LIN {X 0,Y 468.2,Z 260.249,A -85,B 0,C 180,E1 -7618.306,E2 -7618.306} C_VEL
LIN {X 0,Y 467.957,Z 265.306,A -85,B 0,C 180,E1 -7620.584,E2 -7620.584} C_VEL
LIN {X 0,Y 467.636,Z 273.513,A -85,B 0,C 180,E1 -7624.161,E2 -7624.161} C_VEL
LIN {X 0,Y 467.386,Z 281.282,A -85,B 0,C 180,E1 -7627.453,E2 -7627.453} C_VEL
LIN {X 0,Y 467.175,Z 287.892,A -85,B 0,C 180,E1 -7630.215,E2 -7630.215} C_VEL
LIN {X 0,Y 467.029,Z 295.543,A -85,B 0,C 180,E1 -7633.386,E2 -7633.386} C_VEL
LIN {X 0,Y 466.937,Z 298.461,A -85,B 0,C 180,E1 -7634.594,E2 -7634.594} C_VEL
LIN {X 0,Y 469.237,Z 312.548,A -85,B 0,C 180,E1 -7635.056,E2 -7635.056} C_VEL
LIN {X 0,Y 469.965,Z 320.318,A -85,B 0,C 180,E1 -7635.383,E2 -7635.383} C_VEL
LIN {X 0,Y 469.517,Z 331.349,A -85,B 0,C 180,E1 -7635.922,E2 -7635.922} C_VEL
LIN {X 0,Y 469.015,Z 343.205,A -85,B 0,C 180,E1 -7636.68,E2 -7636.68} C_VEL
LIN {X 0,Y 468.525,Z 353.704,A -85,B 0,C 180,E1 -7637.535,E2 -7637.535} C_VEL
LIN {X 0,Y 468.12,Z 363.549,A -85,B 0,C 180,E1 -7638.526,E2 -7638.526} C_VEL
LIN {X 0,Y 467.618,Z 372.397,A -85,B 0,C 180,E1 -7639.61,E2 -7639.61} C_VEL
LIN {X 0,Y 467.263,Z 381.03,A -85,B 0,C 180,E1 -7640.913,E2 -7640.913} C_VEL
LIN {X 0,Y 466.991,Z 387.93,A -85,B 0,C 180,E1 -7642.215,E2 -7642.215} C_VEL
LIN {X 0,Y 466.816,Z 393.538,A -85,B 0,C 180,E1 -7643.537,E2 -7643.537} C_VEL
LIN {X 0,Y 466.737,Z 397.799,A -85,B 0,C 180,E1 -7644.816,E2 -7644.816} C_VEL
LIN {X 0,Y 466.647,Z 400.094,A -85,B 0,C 180,E1 -7645.681,E2 -7645.681} C_VEL
LIN {X 0,Y 466.689,Z 401.958,A -85,B 0,C 180,E1 -7646.546,E2 -7646.546} C_VEL
LIN {X 0,Y 466.662,Z 403.353,A -85,B 0,C 180,E1 -7647.41,E2 -7647.41} C_VEL
LIN {X 0,Y 466.618,Z 404.957,A -85,B 0,C 180,E1 -7649.137,E2 -7649.137} C_VEL
LIN {X 0,Y 466.598,Z 405.173,A -85,B 0,C 180,E1 -7650,E2 -7650} C_VEL
LIN {X 0,Y 466.618,Z 404.957,A -85,B 0,C 180,E1 -7650.863,E2 -7650.863} C_VEL
LIN {X 0,Y 466.662,Z 403.356,A -85,B 0,C 180,E1 -7652.589,E2 -7652.589} C_VEL
LIN {X 0,Y 466.689,Z 401.961,A -85,B 0,C 180,E1 -7653.453,E2 -7653.453} C_VEL
LIN {X 0,Y 466.689,Z 399.024,A -85,B 0,C 180,E1 -7654.751,E2 -7654.751} C_VEL
LIN {X 0,Y 466.755,Z 395.05,A -85,B 0,C 180,E1 -7656.05,E2 -7656.05} C_VEL
LIN {X 0,Y 466.971,Z 388.941,A -85,B 0,C 180,E1 -7657.567,E2 -7657.567} C_VEL
LIN {X 0,Y 467.227,Z 382.264,A -85,B 0,C 180,E1 -7658.869,E2 -7658.869} C_VEL
LIN {X 0,Y 467.565,Z 373.98,A -85,B 0,C 180,E1 -7660.173,E2 -7660.173} C_VEL
LIN {X 0,Y 468.023,Z 365.492,A -85,B 0,C 180,E1 -7661.257,E2 -7661.257} C_VEL
LIN {X 0,Y 468.46,Z 355.447,A -85,B 0,C 180,E1 -7662.303,E2 -7662.303} C_VEL
LIN {X 0,Y 468.941,Z 344.625,A -85,B 0,C 180,E1 -7663.212,E2 -7663.212} C_VEL
LIN {X 0,Y 469.441,Z 333.25,A -85,B 0,C 180,E1 -7663.97,E2 -7663.97} C_VEL
LIN {X 0,Y 469.914,Z 321.583,A -85,B 0,C 180,E1 -7664.563,E2 -7664.563} C_VEL
LIN {X 0,Y 469.724,Z 316.487,A -85,B 0,C 180,E1 -7664.783,E2 -7664.783} C_VEL
LIN {X 0,Y 467.709,Z 303.026,A -85,B 0,C 180,E1 -7665.271,E2 -7665.271} C_VEL
LIN {X 0,Y 466.937,Z 298.457,A -85,B 0,C 180,E1 -7665.406,E2 -7665.406} C_VEL
LIN {X 0,Y 467.114,Z 290.788,A -85,B 0,C 180,E1 -7668.581,E2 -7668.581} C_VEL
LIN {X 0,Y 467.347,Z 283.49,A -85,B 0,C 180,E1 -7671.619,E2 -7671.619} C_VEL
LIN {X 0,Y 467.56,Z 275.713,A -85,B 0,C 180,E1 -7674.89,E2 -7674.89} C_VEL
LIN {X 0,Y 467.794,Z 267.942,A -85,B 0,C 180,E1 -7678.245,E2 -7678.245} C_VEL
LIN {X 0,Y 468.087,Z 262.432,A -85,B 0,C 180,E1 -7680.696,E2 -7680.696} C_VEL
LIN {X 0,Y 468.438,Z 255.839,A -85,B 0,C 180,E1 -7683.719,E2 -7683.719} C_VEL
LIN {X 0,Y 468.486,Z 251.281,A -85,B 0,C 180,E1 -7685.896,E2 -7685.896} C_VEL
LIN {X 0,Y 467.682,Z 245.54,A -85,B 0,C 180,E1 -7688.834,E2 -7688.834} C_VEL
LIN {X 0,Y 467.621,Z 245.24,A -85,B 0,C 180,E1 -7689.141,E2 -7689.141} C_VEL
LIN {X 0,Y 467.588,Z 245.241,A -85,B 0,C 180,E1 -7692.567,E2 -7692.567} C_VEL
LIN {X 0,Y 467.567,Z 245.245,A -85,B 0,C 180,E1 -7695.052,E2 -7695.052} C_VEL
LIN {X 0,Y 467.566,Z 245.246,A -85,B 0,C 180,E1 -7698.725,E2 -7698.725} C_VEL
LIN {X 0,Y 467.562,Z 245.242,A -85,B 0,C 180,E1 -7701.955,E2 -7701.955} C_VEL
LIN {X 0,Y 467.564,Z 245.243,A -85,B 0,C 180,E1 -7705.167,E2 -7705.167} C_VEL
LIN {X 0,Y 467.585,Z 245.241,A -85,B 0,C 180,E1 -7708.26,E2 -7708.26} C_VEL
LIN {X 0,Y 467.555,Z 245.244,A -85,B 0,C 180,E1 -7711.249,E2 -7711.249} C_VEL
LIN {X 0,Y 467.568,Z 245.246,A -85,B 0,C 180,E1 -7714.157,E2 -7714.157} C_VEL
LIN {X 0,Y 467.577,Z 245.239,A -85,B 0,C 180,E1 -7716.996,E2 -7716.996} C_VEL
LIN {X 0,Y 467.625,Z 245.238,A -85,B 0,C 180,E1 -7719.777,E2 -7719.777} C_VEL
LIN {X 0,Y 467.609,Z 245.239,A -85,B 0,C 180,E1 -7722.507,E2 -7722.507} C_VEL
LIN {X 0,Y 467.605,Z 245.238,A -85,B 0,C 180,E1 -7725.196,E2 -7725.196} C_VEL
LIN {X 0,Y 467.657,Z 245.235,A -85,B 0,C 180,E1 -7727.855,E2 -7727.855} C_VEL
LIN {X 0,Y 467.668,Z 245.232,A -85,B 0,C 180,E1 -7731.357,E2 -7731.357} C_VEL
LIN {X 0,Y 467.736,Z 245.221,A -85,B 0,C 180,E1 -7733.963,E2 -7733.963} C_VEL
LIN {X 0,Y 467.861,Z 245.206,A -85,B 0,C 180,E1 -7737.417,E2 -7737.417} C_VEL
LIN {X 0,Y 467.882,Z 245.204,A -85,B 0,C 180,E1 -7740,E2 -7740} C_VEL
LIN {X 0,Y 467.822,Z 245.21,A -85,B 0,C 180,E1 -7742.583,E2 -7742.583} C_VEL
LIN {X 0,Y 467.725,Z 245.22,A -85,B 0,C 180,E1 -7746.038,E2 -7746.038} C_VEL
LIN {X 0,Y 467.673,Z 245.232,A -85,B 0,C 180,E1 -7748.643,E2 -7748.643} C_VEL
LIN {X 0,Y 467.658,Z 245.232,A -85,B 0,C 180,E1 -7752.145,E2 -7752.145} C_VEL
LIN {X 0,Y 467.64,Z 245.233,A -85,B 0,C 180,E1 -7755.695,E2 -7755.695} C_VEL
LIN {X 0,Y 467.623,Z 245.234,A -85,B 0,C 180,E1 -7759.308,E2 -7759.308} C_VEL
LIN {X 0,Y 467.537,Z 245.247,A -85,B 0,C 180,E1 -7762.074,E2 -7762.074} C_VEL
LIN {X 0,Y 467.588,Z 245.24,A -85,B 0,C 180,E1 -7764.888,E2 -7764.888} C_VEL
LIN {X 0,Y 467.621,Z 245.238,A -85,B 0,C 180,E1 -7767.769,E2 -7767.769} C_VEL
LIN {X 0,Y 467.568,Z 245.242,A -85,B 0,C 180,E1 -7771.045,E2 -7771.045} C_VEL
LIN {X 0,Y 467.578,Z 245.244,A -85,B 0,C 180,E1 -7774.24,E2 -7774.24} C_VEL
LIN {X 0,Y 467.545,Z 245.244,A -85,B 0,C 180,E1 -7777.186,E2 -7777.186} C_VEL
LIN {X 0,Y 467.574,Z 245.242,A -85,B 0,C 180,E1 -7780.265,E2 -7780.265} C_VEL
LIN {X 0,Y 467.549,Z 245.245,A -85,B 0,C 180,E1 -7783.745,E2 -7783.745} C_VEL
LIN {X 0,Y 467.533,Z 245.248,A -85,B 0,C 180,E1 -7786.253,E2 -7786.253} C_VEL
LIN {X 0,Y 467.559,Z 245.246,A -85,B 0,C 180,E1 -7789.733,E2 -7789.733} C_VEL
LIN {X 0,Y 467.54,Z 245.248,A -85,B 0,C 180,E1 -7792.815,E2 -7792.815} C_VEL
LIN {X 0,Y 467.465,Z 245.257,A -85,B 0,C 180,E1 -7794.278,E2 -7794.278} C_VEL
LIN {X 0,Y 467.468,Z 246.827,A -85,B 0,C 180,E1 -7795.78,E2 -7795.78} C_VEL
LIN {X 0,Y 467.357,Z 251.614,A -85,B 0,C 180,E1 -7799.251,E2 -7799.251} C_VEL
LIN {X 0,Y 467.182,Z 255.798,A -85,B 0,C 180,E1 -7802.203,E2 -7802.203} C_VEL
LIN {X 0,Y 467.117,Z 259.954,A -85,B 0,C 180,E1 -7805.085,E2 -7805.085} C_VEL
LIN {X 0,Y 466.987,Z 264.104,A -85,B 0,C 180,E1 -7807.899,E2 -7807.899} C_VEL
LIN {X 0,Y 466.904,Z 269.34,A -85,B 0,C 180,E1 -7811.322,E2 -7811.322} C_VEL
LIN {X 0,Y 466.827,Z 273.108,A -85,B 0,C 180,E1 -7813.712,E2 -7813.712} C_VEL
LIN {X 0,Y 466.726,Z 274.503,A -85,B 0,C 180,E1 -7814.089,E2 -7814.089} C_VEL
LIN {X 0,Y 466.338,Z 277.681,A -85,B 0,C 180,E1 -7814.465,E2 -7814.465} C_VEL
LIN {X 0,Y 465.543,Z 283.2,A -85,B 0,C 180,E1 -7814.816,E2 -7814.816} C_VEL
LIN {X 0,Y 463.983,Z 293.781,A -85,B 0,C 180,E1 -7815.189,E2 -7815.189} C_VEL
LIN {X 0,Y 463.138,Z 301.031,A -85,B 0,C 180,E1 -7815.502,E2 -7815.502} C_VEL
LIN {X 0,Y 462.696,Z 312.356,A -85,B 0,C 180,E1 -7816.159,E2 -7816.159} C_VEL
LIN {X 0,Y 462.211,Z 324.024,A -85,B 0,C 180,E1 -7817.04,E2 -7817.04} C_VEL
LIN {X 0,Y 461.626,Z 334.493,A -85,B 0,C 180,E1 -7818.028,E2 -7818.028} C_VEL
LIN {X 0,Y 461.182,Z 343.044,A -85,B 0,C 180,E1 -7819.019,E2 -7819.019} C_VEL
LIN {X 0,Y 460.763,Z 350.92,A -85,B 0,C 180,E1 -7820.119,E2 -7820.119} C_VEL
LIN {X 0,Y 460.321,Z 358.62,A -85,B 0,C 180,E1 -7821.439,E2 -7821.439} C_VEL
LIN {X 0,Y 460.003,Z 365.682,A -85,B 0,C 180,E1 -7822.98,E2 -7822.98} C_VEL
LIN {X 0,Y 459.88,Z 370.386,A -85,B 0,C 180,E1 -7824.299,E2 -7824.299} C_VEL
LIN {X 0,Y 459.679,Z 373.991,A -85,B 0,C 180,E1 -7825.616,E2 -7825.616} C_VEL
LIN {X 0,Y 459.689,Z 375.851,A -85,B 0,C 180,E1 -7826.494,E2 -7826.494} C_VEL
LIN {X 0,Y 459.607,Z 377.256,A -85,B 0,C 180,E1 -7827.371,E2 -7827.371} C_VEL
LIN {X 0,Y 459.523,Z 378.87,A -85,B 0,C 180,E1 -7829.124,E2 -7829.124} C_VEL
LIN {X 0,Y 459.531,Z 379.105,A -85,B 0,C 180,E1 -7830,E2 -7830} C_VEL
LIN {X 0,Y 459.523,Z 378.919,A -85,B 0,C 180,E1 -7830.876,E2 -7830.876} C_VEL
LIN {X 0,Y 459.607,Z 377.369,A -85,B 0,C 180,E1 -7832.629,E2 -7832.629} C_VEL
LIN {X 0,Y 459.688,Z 376.013,A -85,B 0,C 180,E1 -7833.506,E2 -7833.506} C_VEL
LIN {X 0,Y 459.67,Z 373.152,A -85,B 0,C 180,E1 -7834.824,E2 -7834.824} C_VEL
LIN {X 0,Y 459.941,Z 369.265,A -85,B 0,C 180,E1 -7836.14,E2 -7836.14} C_VEL
LIN {X 0,Y 460.051,Z 364.257,A -85,B 0,C 180,E1 -7837.461,E2 -7837.461} C_VEL
LIN {X 0,Y 460.361,Z 357.95,A -85,B 0,C 180,E1 -7838.781,E2 -7838.781} C_VEL
LIN {X 0,Y 460.782,Z 350.052,A -85,B 0,C 180,E1 -7840.102,E2 -7840.102} C_VEL
LIN {X 0,Y 461.299,Z 340.226,A -85,B 0,C 180,E1 -7841.424,E2 -7841.424} C_VEL
LIN {X 0,Y 461.897,Z 329.928,A -85,B 0,C 180,E1 -7842.521,E2 -7842.521} C_VEL
LIN {X 0,Y 462.402,Z 318.607,A -85,B 0,C 180,E1 -7843.489,E2 -7843.489} C_VEL
LIN {X 0,Y 462.943,Z 306.706,A -85,B 0,C 180,E1 -7844.282,E2 -7844.282} C_VEL
LIN {X 0,Y 463.324,Z 294.664,A -85,B 0,C 180,E1 -7844.887,E2 -7844.887} C_VEL
LIN {X 0,Y 462.666,Z 288.508,A -85,B 0,C 180,E1 -7845.158,E2 -7845.158} C_VEL
LIN {X 0,Y 459.907,Z 275.491,A -85,B 0,C 180,E1 -7845.643,E2 -7845.643} C_VEL
LIN {X 0,Y 459.836,Z 274.771,A -85,B 0,C 180,E1 -7845.704,E2 -7845.704} C_VEL
LIN {X 0,Y 459.843,Z 270.048,A -85,B 0,C 180,E1 -7848.721,E2 -7848.721} C_VEL
LIN {X 0,Y 459.908,Z 265.809,A -85,B 0,C 180,E1 -7851.516,E2 -7851.516} C_VEL
LIN {X 0,Y 460.008,Z 261.63,A -85,B 0,C 180,E1 -7854.363,E2 -7854.363} C_VEL
LIN {X 0,Y 460.133,Z 256.956,A -85,B 0,C 180,E1 -7857.639,E2 -7857.639} C_VEL
LIN {X 0,Y 460.231,Z 253.27,A -85,B 0,C 180,E1 -7860.261,E2 -7860.261} C_VEL
LIN {X 0,Y 460.349,Z 249.051,A -85,B 0,C 180,E1 -7863.34,E2 -7863.34} C_VEL
LIN {X 0,Y 460.367,Z 246.221,A -85,B 0,C 180,E1 -7865.459,E2 -7865.459} C_VEL
LIN {X 0,Y 460.499,Z 246.122,A -85,B 0,C 180,E1 -7867.624,E2 -7867.624} C_VEL
LIN {X 0,Y 460.518,Z 246.12,A -85,B 0,C 180,E1 -7871.013,E2 -7871.013} C_VEL
LIN {X 0,Y 460.512,Z 246.122,A -85,B 0,C 180,E1 -7874.59,E2 -7874.59} C_VEL
LIN {X 0,Y 460.506,Z 246.123,A -85,B 0,C 180,E1 -7877.816,E2 -7877.816} C_VEL
LIN {X 0,Y 460.536,Z 246.117,A -85,B 0,C 180,E1 -7881.104,E2 -7881.104} C_VEL
LIN {X 0,Y 460.511,Z 246.12,A -85,B 0,C 180,E1 -7884.554,E2 -7884.554} C_VEL
LIN {X 0,Y 460.532,Z 246.122,A -85,B 0,C 180,E1 -7887.715,E2 -7887.715} C_VEL
LIN {X 0,Y 460.54,Z 246.118,A -85,B 0,C 180,E1 -7890.769,E2 -7890.769} C_VEL
LIN {X 0,Y 460.559,Z 246.116,A -85,B 0,C 180,E1 -7893.734,E2 -7893.734} C_VEL
LIN {X 0,Y 460.548,Z 246.116,A -85,B 0,C 180,E1 -7896.624,E2 -7896.624} C_VEL
LIN {X 0,Y 460.554,Z 246.119,A -85,B 0,C 180,E1 -7899.453,E2 -7899.453} C_VEL
LIN {X 0,Y 460.543,Z 246.117,A -85,B 0,C 180,E1 -7902.229,E2 -7902.229} C_VEL
LIN {X 0,Y 460.565,Z 246.118,A -85,B 0,C 180,E1 -7904.965,E2 -7904.965} C_VEL
LIN {X 0,Y 460.615,Z 246.11,A -85,B 0,C 180,E1 -7908.559,E2 -7908.559} C_VEL
LIN {X 0,Y 460.624,Z 246.11,A -85,B 0,C 180,E1 -7911.224,E2 -7911.224} C_VEL
LIN {X 0,Y 460.693,Z 246.096,A -85,B 0,C 180,E1 -7913.87,E2 -7913.87} C_VEL
LIN {X 0,Y 460.767,Z 246.089,A -85,B 0,C 180,E1 -7917.377,E2 -7917.377} C_VEL
LIN {X 0,Y 460.825,Z 246.083,A -85,B 0,C 180,E1 -7920,E2 -7920} C_VEL
LIN {X 0,Y 460.803,Z 246.086,A -85,B 0,C 180,E1 -7922.622,E2 -7922.622} C_VEL
LIN {X 0,Y 460.703,Z 246.097,A -85,B 0,C 180,E1 -7926.13,E2 -7926.13} C_VEL
LIN {X 0,Y 460.61,Z 246.11,A -85,B 0,C 180,E1 -7928.776,E2 -7928.776} C_VEL
LIN {X 0,Y 460.599,Z 246.112,A -85,B 0,C 180,E1 -7932.435,E2 -7932.435} C_VEL
LIN {X 0,Y 460.604,Z 246.112,A -85,B 0,C 180,E1 -7935.997,E2 -7935.997} C_VEL
LIN {X 0,Y 460.574,Z 246.114,A -85,B 0,C 180,E1 -7938.902,E2 -7938.902} C_VEL
LIN {X 0,Y 460.519,Z 246.12,A -85,B 0,C 180,E1 -7941.486,E2 -7941.486} C_VEL
LIN {X 0,Y 460.52,Z 246.12,A -85,B 0,C 180,E1 -7944.334,E2 -7944.334} C_VEL
LIN {X 0,Y 460.531,Z 246.119,A -85,B 0,C 180,E1 -7947.247,E2 -7947.247} C_VEL
LIN {X 0,Y 460.509,Z 246.123,A -85,B 0,C 180,E1 -7950.24,E2 -7950.24} C_VEL
LIN {X 0,Y 460.532,Z 246.12,A -85,B 0,C 180,E1 -7953.325,E2 -7953.325} C_VEL
LIN {X 0,Y 460.475,Z 246.125,A -85,B 0,C 180,E1 -7956.53,E2 -7956.53} C_VEL
LIN {X 0,Y 460.515,Z 246.12,A -85,B 0,C 180,E1 -7959.864,E2 -7959.864} C_VEL
LIN {X 0,Y 460.482,Z 246.127,A -85,B 0,C 180,E1 -7962.896,E2 -7962.896} C_VEL
LIN {X 0,Y 460.511,Z 246.123,A -85,B 0,C 180,E1 -7965.831,E2 -7965.831} C_VEL
LIN {X 0,Y 460.533,Z 246.121,A -85,B 0,C 180,E1 -7968.989,E2 -7968.989} C_VEL
LIN {X 0,Y 460.605,Z 246.235,A -85,B 0,C 180,E1 -7970.847,E2 -7970.847} C_VEL
LIN {X 0,Y 461.46,Z 251.948,A -85,B 0,C 180,E1 -7973.822,E2 -7973.822} C_VEL
LIN {X 0,Y 461.425,Z 256.864,A -85,B 0,C 180,E1 -7976.225,E2 -7976.225} C_VEL
LIN {X 0,Y 461.058,Z 264.541,A -85,B 0,C 180,E1 -7979.799,E2 -7979.799} C_VEL
LIN {X 0,Y 460.648,Z 272.27,A -85,B 0,C 180,E1 -7983.251,E2 -7983.251} C_VEL
LIN {X 0,Y 460.39,Z 279.379,A -85,B 0,C 180,E1 -7986.337,E2 -7986.337} C_VEL
LIN {X 0,Y 460.204,Z 286.63,A -85,B 0,C 180,E1 -7989.436,E2 -7989.436} C_VEL
LIN {X 0,Y 459.965,Z 294.285,A -85,B 0,C 180,E1 -7992.665,E2 -7992.665} C_VEL
LIN {X 0,Y 459.85,Z 298.232,A -85,B 0,C 180,E1 -7994.333,E2 -7994.333} C_VEL
LIN {X 0,Y 462.417,Z 313.883,A -85,B 0,C 180,E1 -7994.887,E2 -7994.887} C_VEL
LIN {X 0,Y 463.043,Z 321.426,A -85,B 0,C 180,E1 -7995.216,E2 -7995.216} C_VEL
LIN {X 0,Y 462.528,Z 333.073,A -85,B 0,C 180,E1 -7995.817,E2 -7995.817} C_VEL
LIN {X 0,Y 462.02,Z 344.438,A -85,B 0,C 180,E1 -7996.587,E2 -7996.587} C_VEL
LIN {X 0,Y 461.506,Z 355.549,A -85,B 0,C 180,E1 -7997.536,E2 -7997.536} C_VEL
LIN {X 0,Y 461.061,Z 365.301,A -85,B 0,C 180,E1 -7998.57,E2 -7998.57} C_VEL
LIN {X 0,Y 460.522,Z 373.785,A -85,B 0,C 180,E1 -7999.67,E2 -7999.67} C_VEL
LIN {X 0,Y 460.159,Z 382.067,A -85,B 0,C 180,E1 -8000.993,E2 -8000.993} C_VEL
LIN {X 0,Y 459.888,Z 388.743,A -85,B 0,C 180,E1 -8002.315,E2 -8002.315} C_VEL
LIN {X 0,Y 459.671,Z 394.853,A -85,B 0,C 180,E1 -8003.856,E2 -8003.856} C_VEL
LIN {X 0,Y 459.617,Z 398.825,A -85,B 0,C 180,E1 -8005.176,E2 -8005.176} C_VEL
LIN {X 0,Y 459.584,Z 401.758,A -85,B 0,C 180,E1 -8006.493,E2 -8006.493} C_VEL
LIN {X 0,Y 459.584,Z 403.154,A -85,B 0,C 180,E1 -8007.37,E2 -8007.37} C_VEL
LIN {X 0,Y 459.521,Z 404.757,A -85,B 0,C 180,E1 -8009.124,E2 -8009.124} C_VEL
LIN {X 0,Y 459.53,Z 404.974,A -85,B 0,C 180,E1 -8010,E2 -8010} C_VEL
LIN {X 0,Y 459.521,Z 404.757,A -85,B 0,C 180,E1 -8010.876,E2 -8010.876} C_VEL
LIN {X 0,Y 459.584,Z 403.156,A -85,B 0,C 180,E1 -8012.629,E2 -8012.629} C_VEL
LIN {X 0,Y 459.584,Z 401.76,A -85,B 0,C 180,E1 -8013.507,E2 -8013.507} C_VEL
LIN {X 0,Y 459.617,Z 398.824,A -85,B 0,C 180,E1 -8014.824,E2 -8014.824} C_VEL
LIN {X 0,Y 459.714,Z 393.819,A -85,B 0,C 180,E1 -8016.431,E2 -8016.431} C_VEL
LIN {X 0,Y 459.932,Z 387.726,A -85,B 0,C 180,E1 -8017.905,E2 -8017.905} C_VEL
LIN {X 0,Y 460.23,Z 380.824,A -85,B 0,C 180,E1 -8019.227,E2 -8019.227} C_VEL
LIN {X 0,Y 460.602,Z 372.189,A -85,B 0,C 180,E1 -8020.55,E2 -8020.55} C_VEL
LIN {X 0,Y 461.141,Z 363.339,A -85,B 0,C 180,E1 -8021.65,E2 -8021.65} C_VEL
LIN {X 0,Y 461.644,Z 352.452,A -85,B 0,C 180,E1 -8022.752,E2 -8022.752} C_VEL
LIN {X 0,Y 462.148,Z 341.45,A -85,B 0,C 180,E1 -8023.634,E2 -8023.634} C_VEL
LIN {X 0,Y 462.717,Z 329.129,A -85,B 0,C 180,E1 -8024.401,E2 -8024.401} C_VEL
LIN {X 0,Y 462.995,Z 318.768,A -85,B 0,C 180,E1 -8024.898,E2 -8024.898} C_VEL
LIN {X 0,Y 461.197,Z 306.142,A -85,B 0,C 180,E1 -8025.406,E2 -8025.406} C_VEL
LIN {X 0,Y 459.85,Z 298.222,A -85,B 0,C 180,E1 -8025.667,E2 -8025.667} C_VEL
LIN {X 0,Y 460.053,Z 291.009,A -85,B 0,C 180,E1 -8028.712,E2 -8028.712} C_VEL
LIN {X 0,Y 460.299,Z 283.333,A -85,B 0,C 180,E1 -8031.967,E2 -8031.967} C_VEL
LIN {X 0,Y 460.535,Z 275.574,A -85,B 0,C 180,E1 -8035.296,E2 -8035.296} C_VEL
LIN {X 0,Y 460.864,Z 267.822,A -85,B 0,C 180,E1 -8038.709,E2 -8038.709} C_VEL
LIN {X 0,Y 461.147,Z 261.894,A -85,B 0,C 180,E1 -8041.41,E2 -8041.41} C_VEL
LIN {X 0,Y 461.511,Z 254.948,A -85,B 0,C 180,E1 -8044.682,E2 -8044.682} C_VEL
LIN {X 0,Y 461.228,Z 250.3,A -85,B 0,C 180,E1 -8047.005,E2 -8047.005} C_VEL
LIN {X 0,Y 460.572,Z 246.118,A -85,B 0,C 180,E1 -8049.219,E2 -8049.219} C_VEL
LIN {X 0,Y 460.524,Z 246.126,A -85,B 0,C 180,E1 -8052.181,E2 -8052.181} C_VEL
LIN {X 0,Y 460.513,Z 246.125,A -85,B 0,C 180,E1 -8055.411,E2 -8055.411} C_VEL
LIN {X 0,Y 460.519,Z 246.122,A -85,B 0,C 180,E1 -8058.987,E2 -8058.987} C_VEL
LIN {X 0,Y 460.499,Z 246.127,A -85,B 0,C 180,E1 -8062.377,E2 -8062.377} C_VEL
LIN {X 0,Y 460.547,Z 246.117,A -85,B 0,C 180,E1 -8065.624,E2 -8065.624} C_VEL
LIN {X 0,Y 460.539,Z 246.121,A -85,B 0,C 180,E1 -8068.745,E2 -8068.745} C_VEL
LIN {X 0,Y 460.551,Z 246.119,A -85,B 0,C 180,E1 -8072.261,E2 -8072.261} C_VEL
LIN {X 0,Y 460.523,Z 246.119,A -85,B 0,C 180,E1 -8074.703,E2 -8074.703} C_VEL
LIN {X 0,Y 460.512,Z 246.122,A -85,B 0,C 180,E1 -8077.571,E2 -8077.571} C_VEL
LIN {X 0,Y 460.571,Z 246.114,A -85,B 0,C 180,E1 -8080.385,E2 -8080.385} C_VEL
LIN {X 0,Y 460.566,Z 246.116,A -85,B 0,C 180,E1 -8083.146,E2 -8083.146} C_VEL
LIN {X 0,Y 460.553,Z 246.118,A -85,B 0,C 180,E1 -8085.868,E2 -8085.868} C_VEL
LIN {X 0,Y 460.608,Z 246.108,A -85,B 0,C 180,E1 -8088.559,E2 -8088.559} C_VEL
LIN {X 0,Y 460.618,Z 246.109,A -85,B 0,C 180,E1 -8091.224,E2 -8091.224} C_VEL
LIN {X 0,Y 460.701,Z 246.097,A -85,B 0,C 180,E1 -8093.87,E2 -8093.87} C_VEL
LIN {X 0,Y 460.802,Z 246.086,A -85,B 0,C 180,E1 -8097.378,E2 -8097.378} C_VEL
LIN {X 0,Y 460.851,Z 246.079,A -85,B 0,C 180,E1 -8100,E2 -8100} C_VEL
LIN {X 0,Y 460.766,Z 246.089,A -85,B 0,C 180,E1 -8102.623,E2 -8102.623} C_VEL
LIN {X 0,Y 460.692,Z 246.096,A -85,B 0,C 180,E1 -8106.13,E2 -8106.13} C_VEL
LIN {X 0,Y 460.623,Z 246.111,A -85,B 0,C 180,E1 -8108.776,E2 -8108.776} C_VEL
LIN {X 0,Y 460.616,Z 246.111,A -85,B 0,C 180,E1 -8112.445,E2 -8112.445} C_VEL
LIN {X 0,Y 460.602,Z 246.111,A -85,B 0,C 180,E1 -8115.998,E2 -8115.998} C_VEL
LIN {X 0,Y 460.569,Z 246.112,A -85,B 0,C 180,E1 -8119.616,E2 -8119.616} C_VEL
LIN {X 0,Y 460.513,Z 246.124,A -85,B 0,C 180,E1 -8122.429,E2 -8122.429} C_VEL
LIN {X 0,Y 460.555,Z 246.117,A -85,B 0,C 180,E1 -8125.798,E2 -8125.798} C_VEL
LIN {X 0,Y 460.553,Z 246.117,A -85,B 0,C 180,E1 -8128.233,E2 -8128.233} C_VEL
LIN {X 0,Y 460.521,Z 246.12,A -85,B 0,C 180,E1 -8131.283,E2 -8131.283} C_VEL
LIN {X 0,Y 460.523,Z 246.12,A -85,B 0,C 180,E1 -8134.504,E2 -8134.504} C_VEL
LIN {X 0,Y 460.5,Z 246.124,A -85,B 0,C 180,E1 -8137.623,E2 -8137.623} C_VEL
LIN {X 0,Y 460.538,Z 246.118,A -85,B 0,C 180,E1 -8140.269,E2 -8140.269} C_VEL
LIN {X 0,Y 460.51,Z 246.123,A -85,B 0,C 180,E1 -8143.375,E2 -8143.375} C_VEL
LIN {X 0,Y 460.489,Z 246.124,A -85,B 0,C 180,E1 -8146.623,E2 -8146.623} C_VEL
LIN {X 0,Y 460.525,Z 246.122,A -85,B 0,C 180,E1 -8149.733,E2 -8149.733} C_VEL
LIN {X 0,Y 460.496,Z 246.123,A -85,B 0,C 180,E1 -8152.525,E2 -8152.525} C_VEL
LIN {X 0,Y 460.377,Z 246.142,A -85,B 0,C 180,E1 -8154.542,E2 -8154.542} C_VEL
LIN {X 0,Y 460.358,Z 249.508,A -85,B 0,C 180,E1 -8157.104,E2 -8157.104} C_VEL
LIN {X 0,Y 460.259,Z 253.124,A -85,B 0,C 180,E1 -8159.742,E2 -8159.742} C_VEL
LIN {X 0,Y 460.122,Z 257.314,A -85,B 0,C 180,E1 -8162.727,E2 -8162.727} C_VEL
LIN {X 0,Y 460.024,Z 261.487,A -85,B 0,C 180,E1 -8165.639,E2 -8165.639} C_VEL
LIN {X 0,Y 459.912,Z 266.098,A -85,B 0,C 180,E1 -8168.774,E2 -8168.774} C_VEL
LIN {X 0,Y 459.789,Z 271.312,A -85,B 0,C 180,E1 -8172.199,E2 -8172.199} C_VEL
LIN {X 0,Y 459.831,Z 274.824,A -85,B 0,C 180,E1 -8174.421,E2 -8174.421} C_VEL
LIN {X 0,Y 462.871,Z 289.702,A -85,B 0,C 180,E1 -8174.985,E2 -8174.985} C_VEL
LIN {X 0,Y 463.385,Z 293.828,A -85,B 0,C 180,E1 -8175.171,E2 -8175.171} C_VEL
LIN {X 0,Y 463.138,Z 301.031,A -85,B 0,C 180,E1 -8175.502,E2 -8175.502} C_VEL
LIN {X 0,Y 462.242,Z 306.474,A -85,B 0,C 180,E1 -8175.769,E2 -8175.769} C_VEL
LIN {X 0,Y 459.129,Z 315.145,A -85,B 0,C 180,E1 -8176.228,E2 -8176.228} C_VEL
LIN {X 0,Y 455.996,Z 323.415,A -85,B 0,C 180,E1 -8176.783,E2 -8176.783} C_VEL
LIN {X 0,Y 455.073,Z 328.224,A -85,B 0,C 180,E1 -8177.196,E2 -8177.196} C_VEL
LIN {X 0,Y 454.542,Z 337.717,A -85,B 0,C 180,E1 -8178.178,E2 -8178.178} C_VEL
LIN {X 0,Y 454.063,Z 346.563,A -85,B 0,C 180,E1 -8179.296,E2 -8179.296} C_VEL
LIN {X 0,Y 453.545,Z 355.194,A -85,B 0,C 180,E1 -8180.636,E2 -8180.636} C_VEL
LIN {X 0,Y 453.116,Z 362.075,A -85,B 0,C 180,E1 -8181.976,E2 -8181.976} C_VEL
LIN {X 0,Y 452.881,Z 367.544,A -85,B 0,C 180,E1 -8183.306,E2 -8183.306} C_VEL
LIN {X 0,Y 452.699,Z 371.904,A -85,B 0,C 180,E1 -8184.655,E2 -8184.655} C_VEL
LIN {X 0,Y 452.588,Z 374.192,A -85,B 0,C 180,E1 -8185.547,E2 -8185.547} C_VEL
LIN {X 0,Y 452.607,Z 376.052,A -85,B 0,C 180,E1 -8186.439,E2 -8186.439} C_VEL
LIN {X 0,Y 452.534,Z 377.456,A -85,B 0,C 180,E1 -8187.33,E2 -8187.33} C_VEL
LIN {X 0,Y 452.43,Z 379.069,A -85,B 0,C 180,E1 -8189.11,E2 -8189.11} C_VEL
LIN {X 0,Y 452.435,Z 379.304,A -85,B 0,C 180,E1 -8190,E2 -8190} C_VEL
LIN {X 0,Y 452.43,Z 379.118,A -85,B 0,C 180,E1 -8190.89,E2 -8190.89} C_VEL
LIN {X 0,Y 452.534,Z 377.567,A -85,B 0,C 180,E1 -8192.671,E2 -8192.671} C_VEL
LIN {X 0,Y 452.605,Z 376.212,A -85,B 0,C 180,E1 -8193.561,E2 -8193.561} C_VEL
LIN {X 0,Y 452.602,Z 373.351,A -85,B 0,C 180,E1 -8194.899,E2 -8194.899} C_VEL
LIN {X 0,Y 452.88,Z 369.463,A -85,B 0,C 180,E1 -8196.236,E2 -8196.236} C_VEL
LIN {X 0,Y 452.994,Z 364.455,A -85,B 0,C 180,E1 -8197.578,E2 -8197.578} C_VEL
LIN {X 0,Y 453.352,Z 358.147,A -85,B 0,C 180,E1 -8198.918,E2 -8198.918} C_VEL
LIN {X 0,Y 453.778,Z 350.249,A -85,B 0,C 180,E1 -8200.26,E2 -8200.26} C_VEL
LIN {X 0,Y 454.342,Z 340.423,A -85,B 0,C 180,E1 -8201.601,E2 -8201.601} C_VEL
LIN {X 0,Y 454.966,Z 330.264,A -85,B 0,C 180,E1 -8202.702,E2 -8202.702} C_VEL
LIN {X 0,Y 455.514,Z 318.482,A -85,B 0,C 180,E1 -8203.722,E2 -8203.722} C_VEL
LIN {X 0,Y 456.065,Z 306.898,A -85,B 0,C 180,E1 -8204.502,E2 -8204.502} C_VEL
LIN {X 0,Y 456.463,Z 294.853,A -85,B 0,C 180,E1 -8205.117,E2 -8205.117} C_VEL
LIN {X 0,Y 455.176,Z 286.096,A -85,B 0,C 180,E1 -8205.511,E2 -8205.511} C_VEL
LIN {X 0,Y 452.728,Z 275,A -85,B 0,C 180,E1 -8205.932,E2 -8205.932} C_VEL
LIN {X 0,Y 452.78,Z 270.221,A -85,B 0,C 180,E1 -8209.024,E2 -8209.024} C_VEL
LIN {X 0,Y 452.845,Z 265.969,A -85,B 0,C 180,E1 -8211.868,E2 -8211.868} C_VEL
LIN {X 0,Y 452.964,Z 261.776,A -85,B 0,C 180,E1 -8214.767,E2 -8214.767} C_VEL
LIN {X 0,Y 453.079,Z 257.441,A -85,B 0,C 180,E1 -8217.851,E2 -8217.851} C_VEL
LIN {X 0,Y 453.2,Z 253.388,A -85,B 0,C 180,E1 -8220.781,E2 -8220.781} C_VEL
LIN {X 0,Y 453.325,Z 249.149,A -85,B 0,C 180,E1 -8223.926,E2 -8223.926} C_VEL
LIN {X 0,Y 453.346,Z 247.735,A -85,B 0,C 180,E1 -8225.001,E2 -8225.001} C_VEL
LIN {X 0,Y 453.401,Z 247.009,A -85,B 0,C 180,E1 -8226.289,E2 -8226.289} C_VEL
LIN {X 0,Y 453.451,Z 246.998,A -85,B 0,C 180,E1 -8229.454,E2 -8229.454} C_VEL
LIN {X 0,Y 453.44,Z 247.002,A -85,B 0,C 180,E1 -8231.929,E2 -8231.929} C_VEL
LIN {X 0,Y 453.484,Z 246.997,A -85,B 0,C 180,E1 -8235.472,E2 -8235.472} C_VEL
LIN {X 0,Y 453.466,Z 247,A -85,B 0,C 180,E1 -8238.207,E2 -8238.207} C_VEL
LIN {X 0,Y 453.473,Z 246.998,A -85,B 0,C 180,E1 -8240.797,E2 -8240.797} C_VEL
LIN {X 0,Y 453.457,Z 247.002,A -85,B 0,C 180,E1 -8243.917,E2 -8243.917} C_VEL
LIN {X 0,Y 453.481,Z 246.996,A -85,B 0,C 180,E1 -8247.151,E2 -8247.151} C_VEL
LIN {X 0,Y 453.475,Z 246.999,A -85,B 0,C 180,E1 -8250.268,E2 -8250.268} C_VEL
LIN {X 0,Y 453.505,Z 246.995,A -85,B 0,C 180,E1 -8253.294,E2 -8253.294} C_VEL
LIN {X 0,Y 453.501,Z 246.995,A -85,B 0,C 180,E1 -8256.239,E2 -8256.239} C_VEL
LIN {X 0,Y 453.485,Z 246.996,A -85,B 0,C 180,E1 -8259.118,E2 -8259.118} C_VEL
LIN {X 0,Y 453.499,Z 246.994,A -85,B 0,C 180,E1 -8261.944,E2 -8261.944} C_VEL
LIN {X 0,Y 453.536,Z 246.991,A -85,B 0,C 180,E1 -8264.726,E2 -8264.726} C_VEL
LIN {X 0,Y 453.563,Z 246.987,A -85,B 0,C 180,E1 -8268.379,E2 -8268.379} C_VEL
LIN {X 0,Y 453.59,Z 246.985,A -85,B 0,C 180,E1 -8271.087,E2 -8271.087} C_VEL
LIN {X 0,Y 453.661,Z 246.972,A -85,B 0,C 180,E1 -8273.774,E2 -8273.774} C_VEL
LIN {X 0,Y 453.715,Z 246.968,A -85,B 0,C 180,E1 -8277.336,E2 -8277.336} C_VEL
LIN {X 0,Y 453.794,Z 246.958,A -85,B 0,C 180,E1 -8280,E2 -8280} C_VEL
LIN {X 0,Y 453.747,Z 246.965,A -85,B 0,C 180,E1 -8282.663,E2 -8282.663} C_VEL
LIN {X 0,Y 453.67,Z 246.974,A -85,B 0,C 180,E1 -8286.225,E2 -8286.225} C_VEL
LIN {X 0,Y 453.574,Z 246.985,A -85,B 0,C 180,E1 -8288.914,E2 -8288.914} C_VEL
LIN {X 0,Y 453.567,Z 246.987,A -85,B 0,C 180,E1 -8292.529,E2 -8292.529} C_VEL
LIN {X 0,Y 453.548,Z 246.99,A -85,B 0,C 180,E1 -8296.196,E2 -8296.196} C_VEL
LIN {X 0,Y 453.523,Z 246.992,A -85,B 0,C 180,E1 -8299.041,E2 -8299.041} C_VEL
LIN {X 0,Y 453.479,Z 246.998,A -85,B 0,C 180,E1 -8301.836,E2 -8301.836} C_VEL
LIN {X 0,Y 453.472,Z 246.996,A -85,B 0,C 180,E1 -8304.737,E2 -8304.737} C_VEL
LIN {X 0,Y 453.492,Z 246.997,A -85,B 0,C 180,E1 -8307.949,E2 -8307.949} C_VEL
LIN {X 0,Y 453.477,Z 246.997,A -85,B 0,C 180,E1 -8310.76,E2 -8310.76} C_VEL
LIN {X 0,Y 453.479,Z 247,A -85,B 0,C 180,E1 -8313.913,E2 -8313.913} C_VEL
LIN {X 0,Y 453.451,Z 247.001,A -85,B 0,C 180,E1 -8317.19,E2 -8317.19} C_VEL
LIN {X 0,Y 453.472,Z 246.996,A -85,B 0,C 180,E1 -8320.611,E2 -8320.611} C_VEL
LIN {X 0,Y 453.461,Z 247.001,A -85,B 0,C 180,E1 -8324.222,E2 -8324.222} C_VEL
LIN {X 0,Y 453.465,Z 247,A -85,B 0,C 180,E1 -8327.005,E2 -8327.005} C_VEL
LIN {X 0,Y 453.521,Z 247.06,A -85,B 0,C 180,E1 -8330.592,E2 -8330.592} C_VEL
LIN {X 0,Y 454.423,Z 252.561,A -85,B 0,C 180,E1 -8333.535,E2 -8333.535} C_VEL
LIN {X 0,Y 454.469,Z 256.774,A -85,B 0,C 180,E1 -8335.636,E2 -8335.636} C_VEL
LIN {X 0,Y 454.089,Z 263.422,A -85,B 0,C 180,E1 -8338.811,E2 -8338.811} C_VEL
LIN {X 0,Y 453.81,Z 268.83,A -85,B 0,C 180,E1 -8341.309,E2 -8341.309} C_VEL
LIN {X 0,Y 453.471,Z 276.554,A -85,B 0,C 180,E1 -8344.773,E2 -8344.773} C_VEL
LIN {X 0,Y 453.229,Z 284.283,A -85,B 0,C 180,E1 -8348.151,E2 -8348.151} C_VEL
LIN {X 0,Y 452.989,Z 291.243,A -85,B 0,C 180,E1 -8351.156,E2 -8351.156} C_VEL
LIN {X 0,Y 452.809,Z 298.072,A -85,B 0,C 180,E1 -8354.098,E2 -8354.098} C_VEL
LIN {X 0,Y 455.151,Z 312.052,A -85,B 0,C 180,E1 -8354.579,E2 -8354.579} C_VEL
LIN {X 0,Y 456.168,Z 321.232,A -85,B 0,C 180,E1 -8354.988,E2 -8354.988} C_VEL
LIN {X 0,Y 455.626,Z 332.877,A -85,B 0,C 180,E1 -8355.598,E2 -8355.598} C_VEL
LIN {X 0,Y 455.099,Z 344.241,A -85,B 0,C 180,E1 -8356.379,E2 -8356.379} C_VEL
LIN {X 0,Y 454.561,Z 354.121,A -85,B 0,C 180,E1 -8357.224,E2 -8357.224} C_VEL
LIN {X 0,Y 454.129,Z 363.151,A -85,B 0,C 180,E1 -8358.167,E2 -8358.167} C_VEL
LIN {X 0,Y 453.596,Z 372,A -85,B 0,C 180,E1 -8359.285,E2 -8359.285} C_VEL
LIN {X 0,Y 453.199,Z 380.632,A -85,B 0,C 180,E1 -8360.629,E2 -8360.629} C_VEL
LIN {X 0,Y 452.867,Z 387.531,A -85,B 0,C 180,E1 -8361.971,E2 -8361.971} C_VEL
LIN {X 0,Y 452.675,Z 393.063,A -85,B 0,C 180,E1 -8363.314,E2 -8363.314} C_VEL
LIN {X 0,Y 452.566,Z 397.4,A -85,B 0,C 180,E1 -8364.654,E2 -8364.654} C_VEL
LIN {X 0,Y 452.486,Z 399.696,A -85,B 0,C 180,E1 -8365.546,E2 -8365.546} C_VEL
LIN {X 0,Y 452.48,Z 401.558,A -85,B 0,C 180,E1 -8366.438,E2 -8366.438} C_VEL
LIN {X 0,Y 452.508,Z 402.955,A -85,B 0,C 180,E1 -8367.329,E2 -8367.329} C_VEL
LIN {X 0,Y 452.428,Z 404.557,A -85,B 0,C 180,E1 -8369.11,E2 -8369.11} C_VEL
LIN {X 0,Y 452.434,Z 404.774,A -85,B 0,C 180,E1 -8370,E2 -8370} C_VEL
LIN {X 0,Y 452.428,Z 404.557,A -85,B 0,C 180,E1 -8370.89,E2 -8370.89} C_VEL
LIN {X 0,Y 452.508,Z 402.956,A -85,B 0,C 180,E1 -8372.671,E2 -8372.671} C_VEL
LIN {X 0,Y 452.48,Z 401.559,A -85,B 0,C 180,E1 -8373.562,E2 -8373.562} C_VEL
LIN {X 0,Y 452.545,Z 398.623,A -85,B 0,C 180,E1 -8374.9,E2 -8374.9} C_VEL
LIN {X 0,Y 452.61,Z 394.111,A -85,B 0,C 180,E1 -8376.396,E2 -8376.396} C_VEL
LIN {X 0,Y 452.83,Z 388.537,A -85,B 0,C 180,E1 -8377.805,E2 -8377.805} C_VEL
LIN {X 0,Y 453.114,Z 381.859,A -85,B 0,C 180,E1 -8379.148,E2 -8379.148} C_VEL
LIN {X 0,Y 453.502,Z 373.574,A -85,B 0,C 180,E1 -8380.492,E2 -8380.492} C_VEL
LIN {X 0,Y 454.045,Z 365.087,A -85,B 0,C 180,E1 -8381.608,E2 -8381.608} C_VEL
LIN {X 0,Y 454.534,Z 355.45,A -85,B 0,C 180,E1 -8382.646,E2 -8382.646} C_VEL
LIN {X 0,Y 455.084,Z 344.217,A -85,B 0,C 180,E1 -8383.622,E2 -8383.622} C_VEL
LIN {X 0,Y 455.635,Z 332.841,A -85,B 0,C 180,E1 -8384.402,E2 -8384.402} C_VEL
LIN {X 0,Y 456.159,Z 321.171,A -85,B 0,C 180,E1 -8385.012,E2 -8385.012} C_VEL
LIN {X 0,Y 454.63,Z 308.857,A -85,B 0,C 180,E1 -8385.543,E2 -8385.543} C_VEL
LIN {X 0,Y 452.812,Z 298.058,A -85,B 0,C 180,E1 -8385.905,E2 -8385.905} C_VEL
LIN {X 0,Y 452.989,Z 290.835,A -85,B 0,C 180,E1 -8389.015,E2 -8389.015} C_VEL
LIN {X 0,Y 453.261,Z 283.177,A -85,B 0,C 180,E1 -8392.326,E2 -8392.326} C_VEL
LIN {X 0,Y 453.523,Z 275.435,A -85,B 0,C 180,E1 -8395.715,E2 -8395.715} C_VEL
LIN {X 0,Y 453.847,Z 267.698,A -85,B 0,C 180,E1 -8399.195,E2 -8399.195} C_VEL
LIN {X 0,Y 454.213,Z 261.124,A -85,B 0,C 180,E1 -8402.264,E2 -8402.264} C_VEL
LIN {X 0,Y 454.522,Z 255.527,A -85,B 0,C 180,E1 -8404.964,E2 -8404.964} C_VEL
LIN {X 0,Y 454.223,Z 251.292,A -85,B 0,C 180,E1 -8407.116,E2 -8407.116} C_VEL
LIN {X 0,Y 453.531,Z 246.997,A -85,B 0,C 180,E1 -8409.445,E2 -8409.445} C_VEL
LIN {X 0,Y 453.464,Z 247,A -85,B 0,C 180,E1 -8412.995,E2 -8412.995} C_VEL
LIN {X 0,Y 453.46,Z 247.001,A -85,B 0,C 180,E1 -8415.778,E2 -8415.778} C_VEL
LIN {X 0,Y 453.471,Z 246.996,A -85,B 0,C 180,E1 -8419.413,E2 -8419.413} C_VEL
LIN {X 0,Y 453.45,Z 247.001,A -85,B 0,C 180,E1 -8422.81,E2 -8422.81} C_VEL
LIN {X 0,Y 453.478,Z 247,A -85,B 0,C 180,E1 -8426.087,E2 -8426.087} C_VEL
LIN {X 0,Y 453.477,Z 246.998,A -85,B 0,C 180,E1 -8429.24,E2 -8429.24} C_VEL
LIN {X 0,Y 453.508,Z 246.997,A -85,B 0,C 180,E1 -8432.296,E2 -8432.296} C_VEL
LIN {X 0,Y 453.471,Z 246.996,A -85,B 0,C 180,E1 -8435.263,E2 -8435.263} C_VEL
LIN {X 0,Y 453.482,Z 246.997,A -85,B 0,C 180,E1 -8438.415,E2 -8438.415} C_VEL
LIN {X 0,Y 453.524,Z 246.992,A -85,B 0,C 180,E1 -8441.009,E2 -8441.009} C_VEL
LIN {X 0,Y 453.571,Z 246.987,A -85,B 0,C 180,E1 -8443.88,E2 -8443.88} C_VEL
LIN {X 0,Y 453.566,Z 246.987,A -85,B 0,C 180,E1 -8447.471,E2 -8447.471} C_VEL
LIN {X 0,Y 453.584,Z 246.984,A -85,B 0,C 180,E1 -8451.086,E2 -8451.086} C_VEL
LIN {X 0,Y 453.668,Z 246.974,A -85,B 0,C 180,E1 -8453.775,E2 -8453.775} C_VEL
LIN {X 0,Y 453.746,Z 246.965,A -85,B 0,C 180,E1 -8457.337,E2 -8457.337} C_VEL
LIN {X 0,Y 453.821,Z 246.955,A -85,B 0,C 180,E1 -8460,E2 -8460} C_VEL
LIN {X 0,Y 453.714,Z 246.968,A -85,B 0,C 180,E1 -8462.664,E2 -8462.664} C_VEL
LIN {X 0,Y 453.66,Z 246.972,A -85,B 0,C 180,E1 -8466.226,E2 -8466.226} C_VEL
LIN {X 0,Y 453.589,Z 246.986,A -85,B 0,C 180,E1 -8468.914,E2 -8468.914} C_VEL
LIN {X 0,Y 453.566,Z 246.988,A -85,B 0,C 180,E1 -8472.529,E2 -8472.529} C_VEL
LIN {X 0,Y 453.546,Z 246.989,A -85,B 0,C 180,E1 -8476.196,E2 -8476.196} C_VEL
LIN {X 0,Y 453.518,Z 246.993,A -85,B 0,C 180,E1 -8479.039,E2 -8479.039} C_VEL
LIN {X 0,Y 453.478,Z 246.996,A -85,B 0,C 180,E1 -8481.836,E2 -8481.836} C_VEL
LIN {X 0,Y 453.503,Z 246.995,A -85,B 0,C 180,E1 -8484.735,E2 -8484.735} C_VEL
LIN {X 0,Y 453.533,Z 246.992,A -85,B 0,C 180,E1 -8487.959,E2 -8487.959} C_VEL
LIN {X 0,Y 453.465,Z 246.999,A -85,B 0,C 180,E1 -8491.525,E2 -8491.525} C_VEL
LIN {X 0,Y 453.483,Z 246.995,A -85,B 0,C 180,E1 -8494.776,E2 -8494.776} C_VEL
LIN {X 0,Y 453.46,Z 247,A -85,B 0,C 180,E1 -8498.312,E2 -8498.312} C_VEL
LIN {X 0,Y 453.495,Z 246.996,A -85,B 0,C 180,E1 -8500.609,E2 -8500.609} C_VEL
LIN {X 0,Y 453.461,Z 247.002,A -85,B 0,C 180,E1 -8504.222,E2 -8504.222} C_VEL
LIN {X 0,Y 453.417,Z 247.005,A -85,B 0,C 180,E1 -8507,E2 -8507} C_VEL
LIN {X 0,Y 453.471,Z 247,A -85,B 0,C 180,E1 -8509.413,E2 -8509.413} C_VEL
LIN {X 0,Y 453.443,Z 247.004,A -85,B 0,C 180,E1 -8512.809,E2 -8512.809} C_VEL
LIN {X 0,Y 453.397,Z 247.009,A -85,B 0,C 180,E1 -8513.912,E2 -8513.912} C_VEL
LIN {X 0,Y 453.372,Z 247.93,A -85,B 0,C 180,E1 -8515.244,E2 -8515.244} C_VEL
LIN {X 0,Y 453.261,Z 251.84,A -85,B 0,C 180,E1 -8518.185,E2 -8518.185} C_VEL
LIN {X 0,Y 453.149,Z 256.048,A -85,B 0,C 180,E1 -8521.263,E2 -8521.263} C_VEL
LIN {X 0,Y 453.019,Z 260.237,A -85,B 0,C 180,E1 -8524.254,E2 -8524.254} C_VEL
LIN {X 0,Y 452.883,Z 264.414,A -85,B 0,C 180,E1 -8527.172,E2 -8527.172} C_VEL
LIN {X 0,Y 452.772,Z 268.658,A -85,B 0,C 180,E1 -8530.032,E2 -8530.032} C_VEL
LIN {X 0,Y 452.685,Z 272.944,A -85,B 0,C 180,E1 -8532.844,E2 -8532.844} C_VEL
LIN {X 0,Y 452.734,Z 275.022,A -85,B 0,C 180,E1 -8534.176,E2 -8534.176} C_VEL
LIN {X 0,Y 455.557,Z 288.409,A -85,B 0,C 180,E1 -8534.681,E2 -8534.681} C_VEL
LIN {X 0,Y 456.505,Z 295.335,A -85,B 0,C 180,E1 -8534.999,E2 -8534.999} C_VEL
LIN {X 0,Y 456.017,Z 307.265,A -85,B 0,C 180,E1 -8535.61,E2 -8535.61} C_VEL
LIN {X 0,Y 455.511,Z 319.032,A -85,B 0,C 180,E1 -8536.414,E2 -8536.414} C_VEL
LIN {X 0,Y 455.073,Z 328.224,A -85,B 0,C 180,E1 -8537.196,E2 -8537.196} C_VEL
LIN {X 0,Y 454.127,Z 332.974,A -85,B 0,C 180,E1 -8537.64,E2 -8537.64} C_VEL
LIN {X 0,Y 450.87,Z 340.356,A -85,B 0,C 180,E1 -8538.38,E2 -8538.38} C_VEL
LIN {X 0,Y 447.661,Z 347.143,A -85,B 0,C 180,E1 -8539.196,E2 -8539.196} C_VEL
LIN {X 0,Y 446.785,Z 350.966,A -85,B 0,C 180,E1 -8539.751,E2 -8539.751} C_VEL
LIN {X 0,Y 446.364,Z 357.851,A -85,B 0,C 180,E1 -8540.941,E2 -8540.941} C_VEL
LIN {X 0,Y 445.978,Z 364.276,A -85,B 0,C 180,E1 -8542.302,E2 -8542.302} C_VEL
LIN {X 0,Y 445.806,Z 369.37,A -85,B 0,C 180,E1 -8543.664,E2 -8543.664} C_VEL
LIN {X 0,Y 445.544,Z 373.331,A -85,B 0,C 180,E1 -8545.023,E2 -8545.023} C_VEL
LIN {X 0,Y 445.51,Z 376.253,A -85,B 0,C 180,E1 -8546.382,E2 -8546.382} C_VEL
LIN {X 0,Y 445.462,Z 377.656,A -85,B 0,C 180,E1 -8547.287,E2 -8547.287} C_VEL
LIN {X 0,Y 445.341,Z 379.269,A -85,B 0,C 180,E1 -8549.096,E2 -8549.096} C_VEL
LIN {X 0,Y 445.343,Z 379.504,A -85,B 0,C 180,E1 -8550,E2 -8550} C_VEL
LIN {X 0,Y 445.341,Z 379.317,A -85,B 0,C 180,E1 -8550.904,E2 -8550.904} C_VEL
LIN {X 0,Y 445.462,Z 377.766,A -85,B 0,C 180,E1 -8552.713,E2 -8552.713} C_VEL
LIN {X 0,Y 445.508,Z 376.411,A -85,B 0,C 180,E1 -8553.618,E2 -8553.618} C_VEL
LIN {X 0,Y 445.54,Z 373.549,A -85,B 0,C 180,E1 -8554.977,E2 -8554.977} C_VEL
LIN {X 0,Y 445.818,Z 369.662,A -85,B 0,C 180,E1 -8556.336,E2 -8556.336} C_VEL
LIN {X 0,Y 445.963,Z 364.653,A -85,B 0,C 180,E1 -8557.698,E2 -8557.698} C_VEL
LIN {X 0,Y 446.348,Z 358.344,A -85,B 0,C 180,E1 -8559.059,E2 -8559.059} C_VEL
LIN {X 0,Y 446.794,Z 350.446,A -85,B 0,C 180,E1 -8560.422,E2 -8560.422} C_VEL
LIN {X 0,Y 447.387,Z 340.619,A -85,B 0,C 180,E1 -8561.784,E2 -8561.784} C_VEL
LIN {X 0,Y 448.041,Z 330.604,A -85,B 0,C 180,E1 -8562.887,E2 -8562.887} C_VEL
LIN {X 0,Y 448.54,Z 320.098,A -85,B 0,C 180,E1 -8563.824,E2 -8563.824} C_VEL
LIN {X 0,Y 449.111,Z 308.914,A -85,B 0,C 180,E1 -8564.616,E2 -8564.616} C_VEL
LIN {X 0,Y 449.606,Z 296.34,A -85,B 0,C 180,E1 -8565.295,E2 -8565.295} C_VEL
LIN {X 0,Y 448.809,Z 289.683,A -85,B 0,C 180,E1 -8565.608,E2 -8565.608} C_VEL
LIN {X 0,Y 446.09,Z 277.345,A -85,B 0,C 180,E1 -8566.102,E2 -8566.102} C_VEL
LIN {X 0,Y 445.653,Z 275.188,A -85,B 0,C 180,E1 -8566.194,E2 -8566.194} C_VEL
LIN {X 0,Y 445.695,Z 270.396,A -85,B 0,C 180,E1 -8569.338,E2 -8569.338} C_VEL
LIN {X 0,Y 445.784,Z 266.13,A -85,B 0,C 180,E1 -8572.233,E2 -8572.233} C_VEL
LIN {X 0,Y 445.904,Z 261.923,A -85,B 0,C 180,E1 -8575.186,E2 -8575.186} C_VEL
LIN {X 0,Y 446.037,Z 257.733,A -85,B 0,C 180,E1 -8578.21,E2 -8578.21} C_VEL
LIN {X 0,Y 446.155,Z 254.917,A -85,B 0,C 180,E1 -8580.27,E2 -8580.27} C_VEL
LIN {X 0,Y 446.28,Z 250.668,A -85,B 0,C 180,E1 -8583.448,E2 -8583.448} C_VEL
LIN {X 0,Y 446.301,Z 247.895,A -85,B 0,C 180,E1 -8585.637,E2 -8585.637} C_VEL
LIN {X 0,Y 446.412,Z 247.877,A -85,B 0,C 180,E1 -8588.078,E2 -8588.078} C_VEL
LIN {X 0,Y 446.403,Z 247.877,A -85,B 0,C 180,E1 -8591.394,E2 -8591.394} C_VEL
LIN {X 0,Y 446.423,Z 247.877,A -85,B 0,C 180,E1 -8595.108,E2 -8595.108} C_VEL
LIN {X 0,Y 446.421,Z 247.879,A -85,B 0,C 180,E1 -8598.608,E2 -8598.608} C_VEL
LIN {X 0,Y 446.428,Z 247.875,A -85,B 0,C 180,E1 -8600.971,E2 -8600.971} C_VEL
LIN {X 0,Y 446.421,Z 247.877,A -85,B 0,C 180,E1 -8604.374,E2 -8604.374} C_VEL
LIN {X 0,Y 446.422,Z 247.879,A -85,B 0,C 180,E1 -8607.638,E2 -8607.638} C_VEL
LIN {X 0,Y 446.449,Z 247.873,A -85,B 0,C 180,E1 -8610.79,E2 -8610.79} C_VEL
LIN {X 0,Y 446.481,Z 247.871,A -85,B 0,C 180,E1 -8613.848,E2 -8613.848} C_VEL
LIN {X 0,Y 446.43,Z 247.874,A -85,B 0,C 180,E1 -8616.823,E2 -8616.823} C_VEL
LIN {X 0,Y 446.446,Z 247.875,A -85,B 0,C 180,E1 -8619.737,E2 -8619.737} C_VEL
LIN {X 0,Y 446.452,Z 247.872,A -85,B 0,C 180,E1 -8622.597,E2 -8622.597} C_VEL
LIN {X 0,Y 446.469,Z 247.872,A -85,B 0,C 180,E1 -8625.412,E2 -8625.412} C_VEL
LIN {X 0,Y 446.521,Z 247.864,A -85,B 0,C 180,E1 -8628.193,E2 -8628.193} C_VEL
LIN {X 0,Y 446.537,Z 247.863,A -85,B 0,C 180,E1 -8630.945,E2 -8630.945} C_VEL
LIN {X 0,Y 446.631,Z 247.849,A -85,B 0,C 180,E1 -8633.676,E2 -8633.676} C_VEL
LIN {X 0,Y 446.664,Z 247.846,A -85,B 0,C 180,E1 -8637.294,E2 -8637.294} C_VEL
LIN {X 0,Y 446.764,Z 247.834,A -85,B 0,C 180,E1 -8640,E2 -8640} C_VEL
LIN {X 0,Y 446.694,Z 247.844,A -85,B 0,C 180,E1 -8642.705,E2 -8642.705} C_VEL
LIN {X 0,Y 446.638,Z 247.85,A -85,B 0,C 180,E1 -8646.324,E2 -8646.324} C_VEL
LIN {X 0,Y 446.521,Z 247.862,A -85,B 0,C 180,E1 -8649.056,E2 -8649.056} C_VEL
LIN {X 0,Y 446.524,Z 247.864,A -85,B 0,C 180,E1 -8652.73,E2 -8652.73} C_VEL
LIN {X 0,Y 446.493,Z 247.869,A -85,B 0,C 180,E1 -8656.459,E2 -8656.459} C_VEL
LIN {X 0,Y 446.473,Z 247.87,A -85,B 0,C 180,E1 -8659.303,E2 -8659.303} C_VEL
LIN {X 0,Y 446.421,Z 247.88,A -85,B 0,C 180,E1 -8662.199,E2 -8662.199} C_VEL
LIN {X 0,Y 446.424,Z 247.874,A -85,B 0,C 180,E1 -8665.154,E2 -8665.154} C_VEL
LIN {X 0,Y 446.442,Z 247.874,A -85,B 0,C 180,E1 -8668.182,E2 -8668.182} C_VEL
LIN {X 0,Y 446.418,Z 247.879,A -85,B 0,C 180,E1 -8671.3,E2 -8671.3} C_VEL
LIN {X 0,Y 446.431,Z 247.875,A -85,B 0,C 180,E1 -8674.523,E2 -8674.523} C_VEL
LIN {X 0,Y 446.412,Z 247.877,A -85,B 0,C 180,E1 -8678.078,E2 -8678.078} C_VEL
LIN {X 0,Y 446.408,Z 247.881,A -85,B 0,C 180,E1 -8681.393,E2 -8681.393} C_VEL
LIN {X 0,Y 446.453,Z 247.874,A -85,B 0,C 180,E1 -8685.104,E2 -8685.104} C_VEL
LIN {X 0,Y 446.43,Z 247.879,A -85,B 0,C 180,E1 -8688.609,E2 -8688.609} C_VEL
LIN {X 0,Y 446.496,Z 247.938,A -85,B 0,C 180,E1 -8690.363,E2 -8690.363} C_VEL
LIN {X 0,Y 447.362,Z 253.388,A -85,B 0,C 180,E1 -8693.346,E2 -8693.346} C_VEL
LIN {X 0,Y 447.473,Z 257.765,A -85,B 0,C 180,E1 -8695.569,E2 -8695.569} C_VEL
LIN {X 0,Y 447.069,Z 264.316,A -85,B 0,C 180,E1 -8698.75,E2 -8698.75} C_VEL
LIN {X 0,Y 446.665,Z 270.905,A -85,B 0,C 180,E1 -8701.834,E2 -8701.834} C_VEL
LIN {X 0,Y 446.424,Z 277.52,A -85,B 0,C 180,E1 -8704.845,E2 -8704.845} C_VEL
LIN {X 0,Y 446.171,Z 285.352,A -85,B 0,C 180,E1 -8708.335,E2 -8708.335} C_VEL
LIN {X 0,Y 445.861,Z 292.847,A -85,B 0,C 180,E1 -8711.624,E2 -8711.624} C_VEL
LIN {X 0,Y 445.755,Z 297.89,A -85,B 0,C 180,E1 -8713.842,E2 -8713.842} C_VEL
LIN {X 0,Y 448.097,Z 311.849,A -85,B 0,C 180,E1 -8714.33,E2 -8714.33} C_VEL
LIN {X 0,Y 449.248,Z 322.243,A -85,B 0,C 180,E1 -8714.809,E2 -8714.809} C_VEL
LIN {X 0,Y 448.663,Z 334.449,A -85,B 0,C 180,E1 -8715.485,E2 -8715.485} C_VEL
LIN {X 0,Y 447.98,Z 346.895,A -85,B 0,C 180,E1 -8716.389,E2 -8716.389} C_VEL
LIN {X 0,Y 447.412,Z 357.803,A -85,B 0,C 180,E1 -8717.411,E2 -8717.411} C_VEL
LIN {X 0,Y 446.981,Z 366.703,A -85,B 0,C 180,E1 -8718.435,E2 -8718.435} C_VEL
LIN {X 0,Y 446.403,Z 374.878,A -85,B 0,C 180,E1 -8719.569,E2 -8719.569} C_VEL
LIN {X 0,Y 446.016,Z 382.905,A -85,B 0,C 180,E1 -8720.934,E2 -8720.934} C_VEL
LIN {X 0,Y 445.723,Z 389.342,A -85,B 0,C 180,E1 -8722.298,E2 -8722.298} C_VEL
LIN {X 0,Y 445.485,Z 395.326,A -85,B 0,C 180,E1 -8723.936,E2 -8723.936} C_VEL
LIN {X 0,Y 445.412,Z 399.496,A -85,B 0,C 180,E1 -8725.475,E2 -8725.475} C_VEL
LIN {X 0,Y 445.378,Z 401.358,A -85,B 0,C 180,E1 -8726.381,E2 -8726.381} C_VEL
LIN {X 0,Y 445.433,Z 402.756,A -85,B 0,C 180,E1 -8727.287,E2 -8727.287} C_VEL
LIN {X 0,Y 445.338,Z 404.358,A -85,B 0,C 180,E1 -8729.096,E2 -8729.096} C_VEL
LIN {X 0,Y 445.342,Z 404.574,A -85,B 0,C 180,E1 -8730,E2 -8730} C_VEL
LIN {X 0,Y 445.356,Z 403.75,A -85,B 0,C 180,E1 -8731.809,E2 -8731.809} C_VEL
LIN {X 0,Y 445.433,Z 402.757,A -85,B 0,C 180,E1 -8732.713,E2 -8732.713} C_VEL
LIN {X 0,Y 445.378,Z 401.358,A -85,B 0,C 180,E1 -8733.619,E2 -8733.619} C_VEL
LIN {X 0,Y 445.474,Z 398.423,A -85,B 0,C 180,E1 -8734.978,E2 -8734.978} C_VEL
LIN {X 0,Y 445.559,Z 393.015,A -85,B 0,C 180,E1 -8736.748,E2 -8736.748} C_VEL
LIN {X 0,Y 445.799,Z 387.322,A -85,B 0,C 180,E1 -8738.157,E2 -8738.157} C_VEL
LIN {X 0,Y 446.147,Z 380.42,A -85,B 0,C 180,E1 -8739.521,E2 -8739.521} C_VEL
LIN {X 0,Y 446.587,Z 371.784,A -85,B 0,C 180,E1 -8740.885,E2 -8740.885} C_VEL
LIN {X 0,Y 447.168,Z 362.932,A -85,B 0,C 180,E1 -8742.02,E2 -8742.02} C_VEL
LIN {X 0,Y 447.713,Z 352.386,A -85,B 0,C 180,E1 -8743.122,E2 -8743.122} C_VEL
LIN {X 0,Y 448.313,Z 341.042,A -85,B 0,C 180,E1 -8744.063,E2 -8744.063} C_VEL
LIN {X 0,Y 448.971,Z 328.72,A -85,B 0,C 180,E1 -8744.852,E2 -8744.852} C_VEL
LIN {X 0,Y 449.097,Z 319.654,A -85,B 0,C 180,E1 -8745.312,E2 -8745.312} C_VEL
LIN {X 0,Y 447.218,Z 306.226,A -85,B 0,C 180,E1 -8745.884,E2 -8745.884} C_VEL
LIN {X 0,Y 445.754,Z 297.884,A -85,B 0,C 180,E1 -8746.157,E2 -8746.157} C_VEL
LIN {X 0,Y 445.949,Z 290.66,A -85,B 0,C 180,E1 -8749.327,E2 -8749.327} C_VEL
LIN {X 0,Y 446.22,Z 283.019,A -85,B 0,C 180,E1 -8752.698,E2 -8752.698} C_VEL
LIN {X 0,Y 446.459,Z 276.388,A -85,B 0,C 180,E1 -8755.651,E2 -8755.651} C_VEL
LIN {X 0,Y 446.822,Z 268.676,A -85,B 0,C 180,E1 -8759.183,E2 -8759.183} C_VEL
LIN {X 0,Y 447.187,Z 262.108,A -85,B 0,C 180,E1 -8762.3,E2 -8762.3} C_VEL
LIN {X 0,Y 447.521,Z 256.101,A -85,B 0,C 180,E1 -8765.252,E2 -8765.252} C_VEL
LIN {X 0,Y 447.338,Z 253.2,A -85,B 0,C 180,E1 -8766.75,E2 -8766.75} C_VEL
LIN {X 0,Y 446.487,Z 247.874,A -85,B 0,C 180,E1 -8769.685,E2 -8769.685} C_VEL
LIN {X 0,Y 446.43,Z 247.877,A -85,B 0,C 180,E1 -8772.605,E2 -8772.605} C_VEL
LIN {X 0,Y 446.452,Z 247.876,A -85,B 0,C 180,E1 -8775.104,E2 -8775.104} C_VEL
LIN {X 0,Y 446.407,Z 247.881,A -85,B 0,C 180,E1 -8778.606,E2 -8778.606} C_VEL
LIN {X 0,Y 446.411,Z 247.877,A -85,B 0,C 180,E1 -8781.922,E2 -8781.922} C_VEL
LIN {X 0,Y 446.43,Z 247.875,A -85,B 0,C 180,E1 -8785.477,E2 -8785.477} C_VEL
LIN {X 0,Y 446.418,Z 247.879,A -85,B 0,C 180,E1 -8788.7,E2 -8788.7} C_VEL
LIN {X 0,Y 446.449,Z 247.873,A -85,B 0,C 180,E1 -8791.83,E2 -8791.83} C_VEL
LIN {X 0,Y 446.422,Z 247.874,A -85,B 0,C 180,E1 -8794.846,E2 -8794.846} C_VEL
LIN {X 0,Y 446.45,Z 247.873,A -85,B 0,C 180,E1 -8798.245,E2 -8798.245} C_VEL
LIN {X 0,Y 446.459,Z 247.874,A -85,B 0,C 180,E1 -8801.649,E2 -8801.649} C_VEL
LIN {X 0,Y 446.509,Z 247.866,A -85,B 0,C 180,E1 -8804.48,E2 -8804.48} C_VEL
LIN {X 0,Y 446.517,Z 247.864,A -85,B 0,C 180,E1 -8808.193,E2 -8808.193} C_VEL
LIN {X 0,Y 446.531,Z 247.861,A -85,B 0,C 180,E1 -8810.945,E2 -8810.945} C_VEL
LIN {X 0,Y 446.637,Z 247.85,A -85,B 0,C 180,E1 -8813.676,E2 -8813.676} C_VEL
LIN {X 0,Y 446.693,Z 247.844,A -85,B 0,C 180,E1 -8817.295,E2 -8817.295} C_VEL
LIN {X 0,Y 446.791,Z 247.831,A -85,B 0,C 180,E1 -8820,E2 -8820} C_VEL
LIN {X 0,Y 446.663,Z 247.846,A -85,B 0,C 180,E1 -8822.706,E2 -8822.706} C_VEL
LIN {X 0,Y 446.629,Z 247.848,A -85,B 0,C 180,E1 -8826.324,E2 -8826.324} C_VEL
LIN {X 0,Y 446.536,Z 247.863,A -85,B 0,C 180,E1 -8829.055,E2 -8829.055} C_VEL
LIN {X 0,Y 446.523,Z 247.865,A -85,B 0,C 180,E1 -8832.73,E2 -8832.73} C_VEL
LIN {X 0,Y 446.497,Z 247.867,A -85,B 0,C 180,E1 -8836.227,E2 -8836.227} C_VEL
LIN {X 0,Y 446.47,Z 247.869,A -85,B 0,C 180,E1 -8839.303,E2 -8839.303} C_VEL
LIN {X 0,Y 446.42,Z 247.878,A -85,B 0,C 180,E1 -8842.2,E2 -8842.2} C_VEL
LIN {X 0,Y 446.446,Z 247.873,A -85,B 0,C 180,E1 -8845.153,E2 -8845.153} C_VEL
LIN {X 0,Y 446.487,Z 247.87,A -85,B 0,C 180,E1 -8848.179,E2 -8848.179} C_VEL
LIN {X 0,Y 446.416,Z 247.877,A -85,B 0,C 180,E1 -8851.301,E2 -8851.301} C_VEL
LIN {X 0,Y 446.423,Z 247.876,A -85,B 0,C 180,E1 -8854.524,E2 -8854.524} C_VEL
LIN {X 0,Y 446.413,Z 247.879,A -85,B 0,C 180,E1 -8858.079,E2 -8858.079} C_VEL
LIN {X 0,Y 446.424,Z 247.876,A -85,B 0,C 180,E1 -8860.917,E2 -8860.917} C_VEL
LIN {X 0,Y 446.399,Z 247.881,A -85,B 0,C 180,E1 -8863.847,E2 -8863.847} C_VEL
LIN {X 0,Y 446.379,Z 247.881,A -85,B 0,C 180,E1 -8866.406,E2 -8866.406} C_VEL
LIN {X 0,Y 446.4,Z 247.881,A -85,B 0,C 180,E1 -8869.797,E2 -8869.797} C_VEL
LIN {X 0,Y 446.405,Z 247.877,A -85,B 0,C 180,E1 -8872.121,E2 -8872.121} C_VEL
LIN {X 0,Y 446.309,Z 247.893,A -85,B 0,C 180,E1 -8874.364,E2 -8874.364} C_VEL
LIN {X 0,Y 446.305,Z 250.565,A -85,B 0,C 180,E1 -8876.574,E2 -8876.574} C_VEL
LIN {X 0,Y 446.164,Z 255.195,A -85,B 0,C 180,E1 -8880.039,E2 -8880.039} C_VEL
LIN {X 0,Y 446.003,Z 258.988,A -85,B 0,C 180,E1 -8882.808,E2 -8882.808} C_VEL
LIN {X 0,Y 445.885,Z 263.578,A -85,B 0,C 180,E1 -8886.092,E2 -8886.092} C_VEL
LIN {X 0,Y 445.732,Z 268.829,A -85,B 0,C 180,E1 -8889.703,E2 -8889.703} C_VEL
LIN {X 0,Y 445.638,Z 273.131,A -85,B 0,C 180,E1 -8892.564,E2 -8892.564} C_VEL
LIN {X 0,Y 445.686,Z 275.434,A -85,B 0,C 180,E1 -8893.928,E2 -8893.928} C_VEL
LIN {X 0,Y 448.487,Z 288.196,A -85,B 0,C 180,E1 -8894.417,E2 -8894.417} C_VEL
LIN {X 0,Y 449.651,Z 295.545,A -85,B 0,C 180,E1 -8894.765,E2 -8894.765} C_VEL
LIN {X 0,Y 449.148,Z 307.472,A -85,B 0,C 180,E1 -8895.386,E2 -8895.386} C_VEL
LIN {X 0,Y 448.673,Z 318.026,A -85,B 0,C 180,E1 -8896.105,E2 -8896.105} C_VEL
LIN {X 0,Y 448.09,Z 329.484,A -85,B 0,C 180,E1 -8897.097,E2 -8897.097} C_VEL
LIN {X 0,Y 447.445,Z 339.865,A -85,B 0,C 180,E1 -8898.218,E2 -8898.218} C_VEL
LIN {X 0,Y 446.976,Z 348.366,A -85,B 0,C 180,E1 -8899.353,E2 -8899.353} C_VEL
LIN {X 0,Y 446.785,Z 350.966,A -85,B 0,C 180,E1 -8899.751,E2 -8899.751} C_VEL
LIN {X 0,Y 445.911,Z 354.644,A -85,B 0,C 180,E1 -8900.334,E2 -8900.334} C_VEL
LIN {X 0,Y 442.721,Z 360.178,A -85,B 0,C 180,E1 -8901.313,E2 -8901.313} C_VEL
LIN {X 0,Y 439.573,Z 365.129,A -85,B 0,C 180,E1 -8902.358,E2 -8902.358} C_VEL
LIN {X 0,Y 438.774,Z 367.757,A -85,B 0,C 180,E1 -8903.039,E2 -8903.039} C_VEL
LIN {X 0,Y 438.605,Z 372.305,A -85,B 0,C 180,E1 -8904.483,E2 -8904.483} C_VEL
LIN {X 0,Y 438.426,Z 374.594,A -85,B 0,C 180,E1 -8905.403,E2 -8905.403} C_VEL
LIN {X 0,Y 438.414,Z 376.454,A -85,B 0,C 180,E1 -8906.324,E2 -8906.324} C_VEL
LIN {X 0,Y 438.392,Z 377.855,A -85,B 0,C 180,E1 -8907.243,E2 -8907.243} C_VEL
LIN {X 0,Y 438.255,Z 379.469,A -85,B 0,C 180,E1 -8909.081,E2 -8909.081} C_VEL
LIN {X 0,Y 438.254,Z 379.704,A -85,B 0,C 180,E1 -8910,E2 -8910} C_VEL
LIN {X 0,Y 438.255,Z 379.517,A -85,B 0,C 180,E1 -8910.919,E2 -8910.919} C_VEL
LIN {X 0,Y 438.392,Z 377.965,A -85,B 0,C 180,E1 -8912.757,E2 -8912.757} C_VEL
LIN {X 0,Y 438.412,Z 376.611,A -85,B 0,C 180,E1 -8913.677,E2 -8913.677} C_VEL
LIN {X 0,Y 438.482,Z 373.748,A -85,B 0,C 180,E1 -8915.058,E2 -8915.058} C_VEL
LIN {X 0,Y 438.762,Z 369.86,A -85,B 0,C 180,E1 -8916.438,E2 -8916.438} C_VEL
LIN {X 0,Y 438.911,Z 364.852,A -85,B 0,C 180,E1 -8917.823,E2 -8917.823} C_VEL
LIN {X 0,Y 439.319,Z 358.542,A -85,B 0,C 180,E1 -8919.206,E2 -8919.206} C_VEL
LIN {X 0,Y 439.822,Z 350.643,A -85,B 0,C 180,E1 -8920.589,E2 -8920.589} C_VEL
LIN {X 0,Y 440.435,Z 340.815,A -85,B 0,C 180,E1 -8921.973,E2 -8921.973} C_VEL
LIN {X 0,Y 441.119,Z 330.94,A -85,B 0,C 180,E1 -8923.079,E2 -8923.079} C_VEL
LIN {X 0,Y 441.657,Z 320.292,A -85,B 0,C 180,E1 -8924.044,E2 -8924.044} C_VEL
LIN {X 0,Y 442.269,Z 309.107,A -85,B 0,C 180,E1 -8924.847,E2 -8924.847} C_VEL
LIN {X 0,Y 442.761,Z 296.53,A -85,B 0,C 180,E1 -8925.537,E2 -8925.537} C_VEL
LIN {X 0,Y 441.024,Z 286.112,A -85,B 0,C 180,E1 -8926.035,E2 -8926.035} C_VEL
LIN {X 0,Y 438.584,Z 275.39,A -85,B 0,C 180,E1 -8926.456,E2 -8926.456} C_VEL
LIN {X 0,Y 438.64,Z 270.572,A -85,B 0,C 180,E1 -8929.662,E2 -8929.662} C_VEL
LIN {X 0,Y 438.724,Z 266.293,A -85,B 0,C 180,E1 -8932.61,E2 -8932.61} C_VEL
LIN {X 0,Y 438.821,Z 263.474,A -85,B 0,C 180,E1 -8934.608,E2 -8934.608} C_VEL
LIN {X 0,Y 438.948,Z 259.278,A -85,B 0,C 180,E1 -8937.666,E2 -8937.666} C_VEL
LIN {X 0,Y 439.106,Z 255.037,A -85,B 0,C 180,E1 -8940.809,E2 -8940.809} C_VEL
LIN {X 0,Y 439.231,Z 250.774,A -85,B 0,C 180,E1 -8944.058,E2 -8944.058} C_VEL
LIN {X 0,Y 439.257,Z 249.169,A -85,B 0,C 180,E1 -8945.315,E2 -8945.315} C_VEL
LIN {X 0,Y 439.331,Z 248.763,A -85,B 0,C 180,E1 -8946.884,E2 -8946.884} C_VEL
LIN {X 0,Y 439.35,Z 248.755,A -85,B 0,C 180,E1 -8949.841,E2 -8949.841} C_VEL
LIN {X 0,Y 439.336,Z 248.76,A -85,B 0,C 180,E1 -8952.62,E2 -8952.62} C_VEL
LIN {X 0,Y 439.378,Z 248.753,A -85,B 0,C 180,E1 -8955.267,E2 -8955.267} C_VEL
LIN {X 0,Y 439.384,Z 248.754,A -85,B 0,C 180,E1 -8958.744,E2 -8958.744} C_VEL
LIN {X 0,Y 439.372,Z 248.754,A -85,B 0,C 180,E1 -8961.609,E2 -8961.609} C_VEL
LIN {X 0,Y 439.399,Z 248.749,A -85,B 0,C 180,E1 -8964.844,E2 -8964.844} C_VEL
LIN {X 0,Y 439.374,Z 248.755,A -85,B 0,C 180,E1 -8968.139,E2 -8968.139} C_VEL
LIN {X 0,Y 439.435,Z 248.748,A -85,B 0,C 180,E1 -8971.598,E2 -8971.598} C_VEL
LIN {X 0,Y 439.401,Z 248.751,A -85,B 0,C 180,E1 -8974.415,E2 -8974.415} C_VEL
LIN {X 0,Y 439.367,Z 248.756,A -85,B 0,C 180,E1 -8977.425,E2 -8977.425} C_VEL
LIN {X 0,Y 439.444,Z 248.744,A -85,B 0,C 180,E1 -8980.663,E2 -8980.663} C_VEL
LIN {X 0,Y 439.458,Z 248.743,A -85,B 0,C 180,E1 -8984.224,E2 -8984.224} C_VEL
LIN {X 0,Y 439.487,Z 248.74,A -85,B 0,C 180,E1 -8988.001,E2 -8988.001} C_VEL
LIN {X 0,Y 439.5,Z 248.739,A -85,B 0,C 180,E1 -8990.798,E2 -8990.798} C_VEL
LIN {X 0,Y 439.602,Z 248.725,A -85,B 0,C 180,E1 -8993.574,E2 -8993.574} C_VEL
LIN {X 0,Y 439.616,Z 248.724,A -85,B 0,C 180,E1 -8997.251,E2 -8997.251} C_VEL
LIN {X 0,Y 439.713,Z 248.712,A -85,B 0,C 180,E1 -9000,E2 -9000} C_VEL
LIN {X 0,Y 439.644,Z 248.722,A -85,B 0,C 180,E1 -9002.749,E2 -9002.749} C_VEL
LIN {X 0,Y 439.608,Z 248.726,A -85,B 0,C 180,E1 -9006.425,E2 -9006.425} C_VEL
LIN {X 0,Y 439.484,Z 248.738,A -85,B 0,C 180,E1 -9009.202,E2 -9009.202} C_VEL
LIN {X 0,Y 439.468,Z 248.743,A -85,B 0,C 180,E1 -9012.938,E2 -9012.938} C_VEL
LIN {X 0,Y 439.451,Z 248.746,A -85,B 0,C 180,E1 -9016.349,E2 -9016.349} C_VEL
LIN {X 0,Y 439.406,Z 248.751,A -85,B 0,C 180,E1 -9019.626,E2 -9019.626} C_VEL
LIN {X 0,Y 439.366,Z 248.755,A -85,B 0,C 180,E1 -9022.575,E2 -9022.575} C_VEL
LIN {X 0,Y 439.369,Z 248.756,A -85,B 0,C 180,E1 -9025.587,E2 -9025.587} C_VEL
LIN {X 0,Y 439.399,Z 248.75,A -85,B 0,C 180,E1 -9028.675,E2 -9028.675} C_VEL
LIN {X 0,Y 439.373,Z 248.757,A -85,B 0,C 180,E1 -9032.03,E2 -9032.03} C_VEL
LIN {X 0,Y 439.396,Z 248.752,A -85,B 0,C 180,E1 -9035.34,E2 -9035.34} C_VEL
LIN {X 0,Y 439.364,Z 248.753,A -85,B 0,C 180,E1 -9038.597,E2 -9038.597} C_VEL
LIN {X 0,Y 439.36,Z 248.755,A -85,B 0,C 180,E1 -9042.209,E2 -9042.209} C_VEL
LIN {X 0,Y 439.401,Z 248.752,A -85,B 0,C 180,E1 -9045.27,E2 -9045.27} C_VEL
LIN {X 0,Y 439.391,Z 248.756,A -85,B 0,C 180,E1 -9048.743,E2 -9048.743} C_VEL
LIN {X 0,Y 439.445,Z 248.854,A -85,B 0,C 180,E1 -9050.144,E2 -9050.144} C_VEL
LIN {X 0,Y 440.26,Z 253.868,A -85,B 0,C 180,E1 -9052.955,E2 -9052.955} C_VEL
LIN {X 0,Y 440.496,Z 257.658,A -85,B 0,C 180,E1 -9054.944,E2 -9054.944} C_VEL
LIN {X 0,Y 440.143,Z 263.409,A -85,B 0,C 180,E1 -9057.809,E2 -9057.809} C_VEL
LIN {X 0,Y 439.772,Z 269.676,A -85,B 0,C 180,E1 -9060.829,E2 -9060.829} C_VEL
LIN {X 0,Y 439.397,Z 277.377,A -85,B 0,C 180,E1 -9064.414,E2 -9064.414} C_VEL
LIN {X 0,Y 439.138,Z 283.963,A -85,B 0,C 180,E1 -9067.412,E2 -9067.412} C_VEL
LIN {X 0,Y 438.895,Z 290.498,A -85,B 0,C 180,E1 -9070.35,E2 -9070.35} C_VEL
LIN {X 0,Y 438.7,Z 297.684,A -85,B 0,C 180,E1 -9073.566,E2 -9073.566} C_VEL
LIN {X 0,Y 441.214,Z 312.693,A -85,B 0,C 180,E1 -9074.119,E2 -9074.119} C_VEL
LIN {X 0,Y 442.336,Z 323.179,A -85,B 0,C 180,E1 -9074.625,E2 -9074.625} C_VEL
LIN {X 0,Y 441.677,Z 336.022,A -85,B 0,C 180,E1 -9075.368,E2 -9075.368} C_VEL
LIN {X 0,Y 440.983,Z 347.754,A -85,B 0,C 180,E1 -9076.263,E2 -9076.263} C_VEL
LIN {X 0,Y 440.401,Z 358.678,A -85,B 0,C 180,E1 -9077.325,E2 -9077.325} C_VEL
LIN {X 0,Y 439.882,Z 368.292,A -85,B 0,C 180,E1 -9078.48,E2 -9078.48} C_VEL
LIN {X 0,Y 439.325,Z 376.17,A -85,B 0,C 180,E1 -9079.632,E2 -9079.632} C_VEL
LIN {X 0,Y 438.908,Z 383.867,A -85,B 0,C 180,E1 -9081.018,E2 -9081.018} C_VEL
LIN {X 0,Y 438.585,Z 390.965,A -85,B 0,C 180,E1 -9082.635,E2 -9082.635} C_VEL
LIN {X 0,Y 438.384,Z 395.561,A -85,B 0,C 180,E1 -9083.978,E2 -9083.978} C_VEL
LIN {X 0,Y 438.341,Z 399.297,A -85,B 0,C 180,E1 -9085.402,E2 -9085.402} C_VEL
LIN {X 0,Y 438.28,Z 401.158,A -85,B 0,C 180,E1 -9086.322,E2 -9086.322} C_VEL
LIN {X 0,Y 438.341,Z 402.556,A -85,B 0,C 180,E1 -9087.243,E2 -9087.243} C_VEL
LIN {X 0,Y 438.252,Z 404.159,A -85,B 0,C 180,E1 -9089.081,E2 -9089.081} C_VEL
LIN {X 0,Y 438.253,Z 404.375,A -85,B 0,C 180,E1 -9090,E2 -9090} C_VEL
LIN {X 0,Y 438.278,Z 403.551,A -85,B 0,C 180,E1 -9091.838,E2 -9091.838} C_VEL
LIN {X 0,Y 438.341,Z 402.557,A -85,B 0,C 180,E1 -9092.757,E2 -9092.757} C_VEL
LIN {X 0,Y 438.28,Z 401.158,A -85,B 0,C 180,E1 -9093.677,E2 -9093.677} C_VEL
LIN {X 0,Y 438.384,Z 398.222,A -85,B 0,C 180,E1 -9095.058,E2 -9095.058} C_VEL
LIN {X 0,Y 438.448,Z 394.245,A -85,B 0,C 180,E1 -9096.442,E2 -9096.442} C_VEL
LIN {X 0,Y 438.697,Z 388.133,A -85,B 0,C 180,E1 -9098.058,E2 -9098.058} C_VEL
LIN {X 0,Y 439.055,Z 381.455,A -85,B 0,C 180,E1 -9099.443,E2 -9099.443} C_VEL
LIN {X 0,Y 439.497,Z 373.17,A -85,B 0,C 180,E1 -9100.83,E2 -9100.83} C_VEL
LIN {X 0,Y 440.08,Z 364.681,A -85,B 0,C 180,E1 -9101.982,E2 -9101.982} C_VEL
LIN {X 0,Y 440.674,Z 354.801,A -85,B 0,C 180,E1 -9103.075,E2 -9103.075} C_VEL
LIN {X 0,Y 441.264,Z 343.81,A -85,B 0,C 180,E1 -9104.057,E2 -9104.057} C_VEL
LIN {X 0,Y 441.858,Z 332.432,A -85,B 0,C 180,E1 -9104.861,E2 -9104.861} C_VEL
LIN {X 0,Y 442.375,Z 321.972,A -85,B 0,C 180,E1 -9105.433,E2 -9105.433} C_VEL
LIN {X 0,Y 440.657,Z 309.03,A -85,B 0,C 180,E1 -9106.03,E2 -9106.03} C_VEL
LIN {X 0,Y 438.698,Z 297.667,A -85,B 0,C 180,E1 -9106.432,E2 -9106.432} C_VEL
LIN {X 0,Y 438.894,Z 290.483,A -85,B 0,C 180,E1 -9109.65,E2 -9109.65} C_VEL
LIN {X 0,Y 439.138,Z 283.945,A -85,B 0,C 180,E1 -9112.588,E2 -9112.588} C_VEL
LIN {X 0,Y 439.393,Z 277.35,A -85,B 0,C 180,E1 -9115.586,E2 -9115.586} C_VEL
LIN {X 0,Y 439.789,Z 269.654,A -85,B 0,C 180,E1 -9119.17,E2 -9119.17} C_VEL
LIN {X 0,Y 440.142,Z 263.382,A -85,B 0,C 180,E1 -9122.19,E2 -9122.19} C_VEL
LIN {X 0,Y 440.5,Z 257.637,A -85,B 0,C 180,E1 -9125.055,E2 -9125.055} C_VEL
LIN {X 0,Y 440.157,Z 253.313,A -85,B 0,C 180,E1 -9127.355,E2 -9127.355} C_VEL
LIN {X 0,Y 439.429,Z 248.752,A -85,B 0,C 180,E1 -9129.929,E2 -9129.929} C_VEL
LIN {X 0,Y 439.383,Z 248.755,A -85,B 0,C 180,E1 -9132.627,E2 -9132.627} C_VEL
LIN {X 0,Y 439.399,Z 248.754,A -85,B 0,C 180,E1 -9135.27,E2 -9135.27} C_VEL
LIN {X 0,Y 439.358,Z 248.757,A -85,B 0,C 180,E1 -9139.017,E2 -9139.017} C_VEL
LIN {X 0,Y 439.346,Z 248.76,A -85,B 0,C 180,E1 -9142.564,E2 -9142.564} C_VEL
LIN {X 0,Y 439.399,Z 248.752,A -85,B 0,C 180,E1 -9144.844,E2 -9144.844} C_VEL
LIN {X 0,Y 439.375,Z 248.756,A -85,B 0,C 180,E1 -9148.14,E2 -9148.14} C_VEL
LIN {X 0,Y 439.404,Z 248.751,A -85,B 0,C 180,E1 -9151.605,E2 -9151.605} C_VEL
LIN {X 0,Y 439.367,Z 248.756,A -85,B 0,C 180,E1 -9154.413,E2 -9154.413} C_VEL
LIN {X 0,Y 439.365,Z 248.755,A -85,B 0,C 180,E1 -9157.425,E2 -9157.425} C_VEL
LIN {X 0,Y 439.443,Z 248.745,A -85,B 0,C 180,E1 -9160.663,E2 -9160.663} C_VEL
LIN {X 0,Y 439.464,Z 248.745,A -85,B 0,C 180,E1 -9164.225,E2 -9164.225} C_VEL
LIN {X 0,Y 439.484,Z 248.742,A -85,B 0,C 180,E1 -9168.001,E2 -9168.001} C_VEL
LIN {X 0,Y 439.505,Z 248.739,A -85,B 0,C 180,E1 -9171.725,E2 -9171.725} C_VEL
LIN {X 0,Y 439.618,Z 248.723,A -85,B 0,C 180,E1 -9174.496,E2 -9174.496} C_VEL
LIN {X 0,Y 439.635,Z 248.722,A -85,B 0,C 180,E1 -9178.168,E2 -9178.168} C_VEL
LIN {X 0,Y 439.76,Z 248.706,A -85,B 0,C 180,E1 -9180,E2 -9180} C_VEL
LIN {X 0,Y 439.615,Z 248.724,A -85,B 0,C 180,E1 -9182.749,E2 -9182.749} C_VEL
LIN {X 0,Y 439.6,Z 248.725,A -85,B 0,C 180,E1 -9186.426,E2 -9186.426} C_VEL
LIN {X 0,Y 439.499,Z 248.739,A -85,B 0,C 180,E1 -9189.202,E2 -9189.202} C_VEL
LIN {X 0,Y 439.467,Z 248.744,A -85,B 0,C 180,E1 -9192.938,E2 -9192.938} C_VEL
LIN {X 0,Y 439.448,Z 248.746,A -85,B 0,C 180,E1 -9196.348,E2 -9196.348} C_VEL
LIN {X 0,Y 439.404,Z 248.748,A -85,B 0,C 180,E1 -9199.626,E2 -9199.626} C_VEL
LIN {X 0,Y 439.366,Z 248.757,A -85,B 0,C 180,E1 -9202.576,E2 -9202.576} C_VEL
LIN {X 0,Y 439.399,Z 248.751,A -85,B 0,C 180,E1 -9205.585,E2 -9205.585} C_VEL
LIN {X 0,Y 439.419,Z 248.751,A -85,B 0,C 180,E1 -9208.674,E2 -9208.674} C_VEL
LIN {X 0,Y 439.367,Z 248.757,A -85,B 0,C 180,E1 -9212.029,E2 -9212.029} C_VEL
LIN {X 0,Y 439.392,Z 248.75,A -85,B 0,C 180,E1 -9215.34,E2 -9215.34} C_VEL
LIN {X 0,Y 439.371,Z 248.754,A -85,B 0,C 180,E1 -9218.596,E2 -9218.596} C_VEL
LIN {X 0,Y 439.383,Z 248.754,A -85,B 0,C 180,E1 -9221.256,E2 -9221.256} C_VEL
LIN {X 0,Y 439.376,Z 248.754,A -85,B 0,C 180,E1 -9224.733,E2 -9224.733} C_VEL
LIN {X 0,Y 439.348,Z 248.761,A -85,B 0,C 180,E1 -9227.79,E2 -9227.79} C_VEL
LIN {X 0,Y 439.363,Z 248.759,A -85,B 0,C 180,E1 -9231.403,E2 -9231.403} C_VEL
LIN {X 0,Y 439.305,Z 248.765,A -85,B 0,C 180,E1 -9233.706,E2 -9233.706} C_VEL
LIN {X 0,Y 439.29,Z 249.221,A -85,B 0,C 180,E1 -9234.834,E2 -9234.834} C_VEL
LIN {X 0,Y 439.185,Z 253.331,A -85,B 0,C 180,E1 -9238.009,E2 -9238.009} C_VEL
LIN {X 0,Y 439.09,Z 256.302,A -85,B 0,C 180,E1 -9240.252,E2 -9240.252} C_VEL
LIN {X 0,Y 438.912,Z 261.024,A -85,B 0,C 180,E1 -9243.727,E2 -9243.727} C_VEL
LIN {X 0,Y 438.799,Z 264.729,A -85,B 0,C 180,E1 -9246.396,E2 -9246.396} C_VEL
LIN {X 0,Y 438.662,Z 269.001,A -85,B 0,C 180,E1 -9249.361,E2 -9249.361} C_VEL
LIN {X 0,Y 438.569,Z 273.316,A -85,B 0,C 180,E1 -9252.274,E2 -9252.274} C_VEL
LIN {X 0,Y 438.562,Z 275.402,A -85,B 0,C 180,E1 -9253.646,E2 -9253.646} C_VEL
LIN {X 0,Y 441.609,Z 289.217,A -85,B 0,C 180,E1 -9254.2,E2 -9254.2} C_VEL
LIN {X 0,Y 442.766,Z 297.05,A -85,B 0,C 180,E1 -9254.581,E2 -9254.581} C_VEL
LIN {X 0,Y 442.209,Z 309.467,A -85,B 0,C 180,E1 -9255.269,E2 -9255.269} C_VEL
LIN {X 0,Y 441.67,Z 320.722,A -85,B 0,C 180,E1 -9256.086,E2 -9256.086} C_VEL
LIN {X 0,Y 441.026,Z 331.897,A -85,B 0,C 180,E1 -9257.109,E2 -9257.109} C_VEL
LIN {X 0,Y 440.384,Z 341.88,A -85,B 0,C 180,E1 -9258.26,E2 -9258.26} C_VEL
LIN {X 0,Y 439.772,Z 351.529,A -85,B 0,C 180,E1 -9259.643,E2 -9259.643} C_VEL
LIN {X 0,Y 439.254,Z 359.227,A -85,B 0,C 180,E1 -9261.025,E2 -9261.025} C_VEL
LIN {X 0,Y 438.851,Z 366.287,A -85,B 0,C 180,E1 -9262.639,E2 -9262.639} C_VEL
LIN {X 0,Y 438.774,Z 367.757,A -85,B 0,C 180,E1 -9263.039,E2 -9263.039} C_VEL
LIN {X 0,Y 437.994,Z 370.192,A -85,B 0,C 180,E1 -9263.735,E2 -9263.735} C_VEL
LIN {X 0,Y 434.959,Z 373.605,A -85,B 0,C 180,E1 -9264.891,E2 -9264.891} C_VEL
LIN {X 0,Y 432.45,Z 375.816,A -85,B 0,C 180,E1 -9265.847,E2 -9265.847} C_VEL
LIN {X 0,Y 431.389,Z 377.186,A -85,B 0,C 180,E1 -9266.6,E2 -9266.6} C_VEL
LIN {X 0,Y 431.309,Z 377.544,A -85,B 0,C 180,E1 -9266.857,E2 -9266.857} C_VEL
LIN {X 0,Y 431.225,Z 379.053,A -85,B 0,C 180,E1 -9268.132,E2 -9268.132} C_VEL
LIN {X 0,Y 431.168,Z 379.903,A -85,B 0,C 180,E1 -9270,E2 -9270} C_VEL
LIN {X 0,Y 431.172,Z 379.716,A -85,B 0,C 180,E1 -9270.934,E2 -9270.934} C_VEL
LIN {X 0,Y 431.323,Z 378.163,A -85,B 0,C 180,E1 -9272.802,E2 -9272.802} C_VEL
LIN {X 0,Y 431.317,Z 376.81,A -85,B 0,C 180,E1 -9273.737,E2 -9273.737} C_VEL
LIN {X 0,Y 431.428,Z 373.946,A -85,B 0,C 180,E1 -9275.14,E2 -9275.14} C_VEL
LIN {X 0,Y 431.707,Z 369.387,A -85,B 0,C 180,E1 -9276.755,E2 -9276.755} C_VEL
LIN {X 0,Y 431.986,Z 363.079,A -85,B 0,C 180,E1 -9278.42,E2 -9278.42} C_VEL
LIN {X 0,Y 432.46,Z 356.292,A -85,B 0,C 180,E1 -9279.825,E2 -9279.825} C_VEL
LIN {X 0,Y 433.016,Z 347.816,A -85,B 0,C 180,E1 -9281.231,E2 -9281.231} C_VEL
LIN {X 0,Y 433.633,Z 339.098,A -85,B 0,C 180,E1 -9282.401,E2 -9282.401} C_VEL
LIN {X 0,Y 434.302,Z 329.497,A -85,B 0,C 180,E1 -9283.454,E2 -9283.454} C_VEL
LIN {X 0,Y 434.846,Z 319.059,A -85,B 0,C 180,E1 -9284.388,E2 -9284.388} C_VEL
LIN {X 0,Y 435.505,Z 307.473,A -85,B 0,C 180,E1 -9285.203,E2 -9285.203} C_VEL
LIN {X 0,Y 435.881,Z 296.721,A -85,B 0,C 180,E1 -9285.789,E2 -9285.789} C_VEL
LIN {X 0,Y 433.645,Z 284.765,A -85,B 0,C 180,E1 -9286.367,E2 -9286.367} C_VEL
LIN {X 0,Y 431.493,Z 275.566,A -85,B 0,C 180,E1 -9286.744,E2 -9286.744} C_VEL
LIN {X 0,Y 431.585,Z 270.75,A -85,B 0,C 180,E1 -9289.997,E2 -9289.997} C_VEL
LIN {X 0,Y 431.676,Z 266.456,A -85,B 0,C 180,E1 -9293.001,E2 -9293.001} C_VEL
LIN {X 0,Y 431.83,Z 262.231,A -85,B 0,C 180,E1 -9296.067,E2 -9296.067} C_VEL
LIN {X 0,Y 431.976,Z 257.995,A -85,B 0,C 180,E1 -9299.215,E2 -9299.215} C_VEL
LIN {X 0,Y 432.112,Z 253.748,A -85,B 0,C 180,E1 -9302.461,E2 -9302.461} C_VEL
LIN {X 0,Y 432.221,Z 250.885,A -85,B 0,C 180,E1 -9304.688,E2 -9304.688} C_VEL
LIN {X 0,Y 432.207,Z 249.65,A -85,B 0,C 180,E1 -9305.831,E2 -9305.831} C_VEL
LIN {X 0,Y 432.327,Z 249.635,A -85,B 0,C 180,E1 -9308.712,E2 -9308.712} C_VEL
LIN {X 0,Y 432.306,Z 249.634,A -85,B 0,C 180,E1 -9311.801,E2 -9311.801} C_VEL
LIN {X 0,Y 432.335,Z 249.633,A -85,B 0,C 180,E1 -9314.347,E2 -9314.347} C_VEL
LIN {X 0,Y 432.319,Z 249.633,A -85,B 0,C 180,E1 -9317.016,E2 -9317.016} C_VEL
LIN {X 0,Y 432.334,Z 249.632,A -85,B 0,C 180,E1 -9319.821,E2 -9319.821} C_VEL
LIN {X 0,Y 432.309,Z 249.632,A -85,B 0,C 180,E1 -9323.022,E2 -9323.022} C_VEL
LIN {X 0,Y 432.36,Z 249.631,A -85,B 0,C 180,E1 -9325.997,E2 -9325.997} C_VEL
LIN {X 0,Y 432.349,Z 249.631,A -85,B 0,C 180,E1 -9329.49,E2 -9329.49} C_VEL
LIN {X 0,Y 432.393,Z 249.623,A -85,B 0,C 180,E1 -9332.928,E2 -9332.928} C_VEL
LIN {X 0,Y 432.371,Z 249.628,A -85,B 0,C 180,E1 -9336.023,E2 -9336.023} C_VEL
LIN {X 0,Y 432.353,Z 249.628,A -85,B 0,C 180,E1 -9339.046,E2 -9339.046} C_VEL
LIN {X 0,Y 432.359,Z 249.628,A -85,B 0,C 180,E1 -9342.01,E2 -9342.01} C_VEL
LIN {X 0,Y 432.392,Z 249.626,A -85,B 0,C 180,E1 -9344.926,E2 -9344.926} C_VEL
LIN {X 0,Y 432.463,Z 249.616,A -85,B 0,C 180,E1 -9347.803,E2 -9347.803} C_VEL
LIN {X 0,Y 432.467,Z 249.615,A -85,B 0,C 180,E1 -9351.59,E2 -9351.59} C_VEL
LIN {X 0,Y 432.587,Z 249.598,A -85,B 0,C 180,E1 -9354.406,E2 -9354.406} C_VEL
LIN {X 0,Y 432.601,Z 249.597,A -85,B 0,C 180,E1 -9358.138,E2 -9358.138} C_VEL
LIN {X 0,Y 432.663,Z 249.59,A -85,B 0,C 180,E1 -9360,E2 -9360} C_VEL
LIN {X 0,Y 432.595,Z 249.6,A -85,B 0,C 180,E1 -9362.794,E2 -9362.794} C_VEL
LIN {X 0,Y 432.595,Z 249.598,A -85,B 0,C 180,E1 -9365.594,E2 -9365.594} C_VEL
LIN {X 0,Y 432.463,Z 249.617,A -85,B 0,C 180,E1 -9368.41,E2 -9368.41} C_VEL
LIN {X 0,Y 432.456,Z 249.619,A -85,B 0,C 180,E1 -9372.197,E2 -9372.197} C_VEL
LIN {X 0,Y 432.434,Z 249.621,A -85,B 0,C 180,E1 -9376.039,E2 -9376.039} C_VEL
LIN {X 0,Y 432.39,Z 249.624,A -85,B 0,C 180,E1 -9379.485,E2 -9379.485} C_VEL
LIN {X 0,Y 432.315,Z 249.631,A -85,B 0,C 180,E1 -9382.965,E2 -9382.965} C_VEL
LIN {X 0,Y 432.322,Z 249.634,A -85,B 0,C 180,E1 -9386.035,E2 -9386.035} C_VEL
LIN {X 0,Y 432.334,Z 249.631,A -85,B 0,C 180,E1 -9389.188,E2 -9389.188} C_VEL
LIN {X 0,Y 432.326,Z 249.632,A -85,B 0,C 180,E1 -9392.443,E2 -9392.443} C_VEL
LIN {X 0,Y 432.346,Z 249.632,A -85,B 0,C 180,E1 -9395.632,E2 -9395.632} C_VEL
LIN {X 0,Y 432.327,Z 249.63,A -85,B 0,C 180,E1 -9398.712,E2 -9398.712} C_VEL
LIN {X 0,Y 432.311,Z 249.634,A -85,B 0,C 180,E1 -9401.8,E2 -9401.8} C_VEL
LIN {X 0,Y 432.335,Z 249.634,A -85,B 0,C 180,E1 -9404.347,E2 -9404.347} C_VEL
LIN {X 0,Y 432.322,Z 249.634,A -85,B 0,C 180,E1 -9407.016,E2 -9407.016} C_VEL
LIN {X 0,Y 432.382,Z 249.721,A -85,B 0,C 180,E1 -9409.893,E2 -9409.893} C_VEL
LIN {X 0,Y 433.295,Z 255.39,A -85,B 0,C 180,E1 -9413.12,E2 -9413.12} C_VEL
LIN {X 0,Y 433.473,Z 259.735,A -85,B 0,C 180,E1 -9415.426,E2 -9415.426} C_VEL
LIN {X 0,Y 433.014,Z 266.276,A -85,B 0,C 180,E1 -9418.71,E2 -9418.71} C_VEL
LIN {X 0,Y 432.581,Z 272.838,A -85,B 0,C 180,E1 -9421.891,E2 -9421.891} C_VEL
LIN {X 0,Y 432.325,Z 279.427,A -85,B 0,C 180,E1 -9424.997,E2 -9424.997} C_VEL
LIN {X 0,Y 432.011,Z 287.062,A -85,B 0,C 180,E1 -9428.529,E2 -9428.529} C_VEL
LIN {X 0,Y 431.682,Z 294.623,A -85,B 0,C 180,E1 -9431.981,E2 -9431.981} C_VEL
LIN {X 0,Y 431.649,Z 297.639,A -85,B 0,C 180,E1 -9433.308,E2 -9433.308} C_VEL
LIN {X 0,Y 433.883,Z 310.612,A -85,B 0,C 180,E1 -9433.77,E2 -9433.77} C_VEL
LIN {X 0,Y 435.488,Z 322.985,A -85,B 0,C 180,E1 -9434.377,E2 -9434.377} C_VEL
LIN {X 0,Y 434.791,Z 335.826,A -85,B 0,C 180,E1 -9435.131,E2 -9435.131} C_VEL
LIN {X 0,Y 434.169,Z 346.501,A -85,B 0,C 180,E1 -9435.947,E2 -9435.947} C_VEL
LIN {X 0,Y 433.48,Z 357.407,A -85,B 0,C 180,E1 -9437,E2 -9437} C_VEL
LIN {X 0,Y 432.999,Z 366.306,A -85,B 0,C 180,E1 -9438.056,E2 -9438.056} C_VEL
LIN {X 0,Y 432.287,Z 375.97,A -85,B 0,C 180,E1 -9439.461,E2 -9439.461} C_VEL
LIN {X 0,Y 431.857,Z 383.668,A -85,B 0,C 180,E1 -9440.87,E2 -9440.87} C_VEL
LIN {X 0,Y 431.52,Z 390.766,A -85,B 0,C 180,E1 -9442.513,E2 -9442.513} C_VEL
LIN {X 0,Y 431.284,Z 395.793,A -85,B 0,C 180,E1 -9444.02,E2 -9444.02} C_VEL
LIN {X 0,Y 431.271,Z 399.098,A -85,B 0,C 180,E1 -9445.326,E2 -9445.326} C_VEL
LIN {X 0,Y 431.187,Z 400.959,A -85,B 0,C 180,E1 -9446.262,E2 -9446.262} C_VEL
LIN {X 0,Y 431.236,Z 402.357,A -85,B 0,C 180,E1 -9447.197,E2 -9447.197} C_VEL
LIN {X 0,Y 431.203,Z 403.352,A -85,B 0,C 180,E1 -9448.132,E2 -9448.132} C_VEL
LIN {X 0,Y 431.167,Z 404.175,A -85,B 0,C 180,E1 -9450,E2 -9450} C_VEL
LIN {X 0,Y 431.203,Z 403.351,A -85,B 0,C 180,E1 -9451.868,E2 -9451.868} C_VEL
LIN {X 0,Y 431.236,Z 402.356,A -85,B 0,C 180,E1 -9452.802,E2 -9452.802} C_VEL
LIN {X 0,Y 431.187,Z 400.957,A -85,B 0,C 180,E1 -9453.738,E2 -9453.738} C_VEL
LIN {X 0,Y 431.295,Z 398.021,A -85,B 0,C 180,E1 -9455.142,E2 -9455.142} C_VEL
LIN {X 0,Y 431.376,Z 394.044,A -85,B 0,C 180,E1 -9456.548,E2 -9456.548} C_VEL
LIN {X 0,Y 431.634,Z 387.931,A -85,B 0,C 180,E1 -9458.191,E2 -9458.191} C_VEL
LIN {X 0,Y 432.002,Z 381.253,A -85,B 0,C 180,E1 -9459.599,E2 -9459.599} C_VEL
LIN {X 0,Y 432.477,Z 372.966,A -85,B 0,C 180,E1 -9461.008,E2 -9461.008} C_VEL
LIN {X 0,Y 433.121,Z 364.478,A -85,B 0,C 180,E1 -9462.178,E2 -9462.178} C_VEL
LIN {X 0,Y 433.748,Z 353.634,A -85,B 0,C 180,E1 -9463.385,E2 -9463.385} C_VEL
LIN {X 0,Y 434.434,Z 342.176,A -85,B 0,C 180,E1 -9464.402,E2 -9464.402} C_VEL
LIN {X 0,Y 435.136,Z 330.302,A -85,B 0,C 180,E1 -9465.216,E2 -9465.216} C_VEL
LIN {X 0,Y 435.347,Z 321.761,A -85,B 0,C 180,E1 -9465.688,E2 -9465.688} C_VEL
LIN {X 0,Y 433.58,Z 308.629,A -85,B 0,C 180,E1 -9466.305,E2 -9466.305} C_VEL
LIN {X 0,Y 431.663,Z 297.484,A -85,B 0,C 180,E1 -9466.704,E2 -9466.704} C_VEL
LIN {X 0,Y 431.876,Z 289.216,A -85,B 0,C 180,E1 -9470.48,E2 -9470.48} C_VEL
LIN {X 0,Y 432.144,Z 282.699,A -85,B 0,C 180,E1 -9473.481,E2 -9473.481} C_VEL
LIN {X 0,Y 432.357,Z 277.203,A -85,B 0,C 180,E1 -9476.033,E2 -9476.033} C_VEL
LIN {X 0,Y 432.828,Z 269.521,A -85,B 0,C 180,E1 -9479.686,E2 -9479.686} C_VEL
LIN {X 0,Y 433.153,Z 263.884,A -85,B 0,C 180,E1 -9482.466,E2 -9482.466} C_VEL
LIN {X 0,Y 433.492,Z 258.633,A -85,B 0,C 180,E1 -9485.138,E2 -9485.138} C_VEL
LIN {X 0,Y 433.168,Z 254.562,A -85,B 0,C 180,E1 -9487.344,E2 -9487.344} C_VEL
LIN {X 0,Y 432.366,Z 249.632,A -85,B 0,C 180,E1 -9490.184,E2 -9490.184} C_VEL
LIN {X 0,Y 432.318,Z 249.635,A -85,B 0,C 180,E1 -9493.061,E2 -9493.061} C_VEL
LIN {X 0,Y 432.334,Z 249.633,A -85,B 0,C 180,E1 -9495.665,E2 -9495.665} C_VEL
LIN {X 0,Y 432.312,Z 249.635,A -85,B 0,C 180,E1 -9498.401,E2 -9498.401} C_VEL
LIN {X 0,Y 432.33,Z 249.63,A -85,B 0,C 180,E1 -9501.849,E2 -9501.849} C_VEL
LIN {X 0,Y 432.34,Z 249.63,A -85,B 0,C 180,E1 -9505.323,E2 -9505.323} C_VEL
LIN {X 0,Y 432.323,Z 249.635,A -85,B 0,C 180,E1 -9508.654,E2 -9508.654} C_VEL
LIN {X 0,Y 432.344,Z 249.631,A -85,B 0,C 180,E1 -9511.874,E2 -9511.874} C_VEL
LIN {X 0,Y 432.324,Z 249.63,A -85,B 0,C 180,E1 -9514.997,E2 -9514.997} C_VEL
LIN {X 0,Y 432.359,Z 249.63,A -85,B 0,C 180,E1 -9518.046,E2 -9518.046} C_VEL
LIN {X 0,Y 432.388,Z 249.624,A -85,B 0,C 180,E1 -9521.03,E2 -9521.03} C_VEL
LIN {X 0,Y 432.432,Z 249.621,A -85,B 0,C 180,E1 -9523.961,E2 -9523.961} C_VEL
LIN {X 0,Y 432.46,Z 249.619,A -85,B 0,C 180,E1 -9527.803,E2 -9527.803} C_VEL
LIN {X 0,Y 432.465,Z 249.618,A -85,B 0,C 180,E1 -9531.59,E2 -9531.59} C_VEL
LIN {X 0,Y 432.594,Z 249.598,A -85,B 0,C 180,E1 -9534.406,E2 -9534.406} C_VEL
LIN {X 0,Y 432.605,Z 249.597,A -85,B 0,C 180,E1 -9538.138,E2 -9538.138} C_VEL
LIN {X 0,Y 432.729,Z 249.582,A -85,B 0,C 180,E1 -9540,E2 -9540} C_VEL
LIN {X 0,Y 432.568,Z 249.602,A -85,B 0,C 180,E1 -9542.794,E2 -9542.794} C_VEL
LIN {X 0,Y 432.586,Z 249.599,A -85,B 0,C 180,E1 -9545.594,E2 -9545.594} C_VEL
LIN {X 0,Y 432.466,Z 249.615,A -85,B 0,C 180,E1 -9548.41,E2 -9548.41} C_VEL
LIN {X 0,Y 432.461,Z 249.616,A -85,B 0,C 180,E1 -9552.197,E2 -9552.197} C_VEL
LIN {X 0,Y 432.431,Z 249.619,A -85,B 0,C 180,E1 -9556.039,E2 -9556.039} C_VEL
LIN {X 0,Y 432.388,Z 249.622,A -85,B 0,C 180,E1 -9559.485,E2 -9559.485} C_VEL
LIN {X 0,Y 432.32,Z 249.633,A -85,B 0,C 180,E1 -9562.964,E2 -9562.964} C_VEL
LIN {X 0,Y 432.363,Z 249.63,A -85,B 0,C 180,E1 -9566.033,E2 -9566.033} C_VEL
LIN {X 0,Y 432.344,Z 249.629,A -85,B 0,C 180,E1 -9569.188,E2 -9569.188} C_VEL
LIN {X 0,Y 432.322,Z 249.635,A -85,B 0,C 180,E1 -9572.443,E2 -9572.443} C_VEL
LIN {X 0,Y 432.337,Z 249.632,A -85,B 0,C 180,E1 -9575.818,E2 -9575.818} C_VEL
LIN {X 0,Y 432.323,Z 249.633,A -85,B 0,C 180,E1 -9579.346,E2 -9579.346} C_VEL
LIN {X 0,Y 432.326,Z 249.634,A -85,B 0,C 180,E1 -9581.798,E2 -9581.798} C_VEL
LIN {X 0,Y 432.333,Z 249.632,A -85,B 0,C 180,E1 -9584.348,E2 -9584.348} C_VEL
LIN {X 0,Y 432.301,Z 249.635,A -85,B 0,C 180,E1 -9587.019,E2 -9587.019} C_VEL
LIN {X 0,Y 432.291,Z 249.638,A -85,B 0,C 180,E1 -9589.828,E2 -9589.828} C_VEL
LIN {X 0,Y 432.312,Z 249.637,A -85,B 0,C 180,E1 -9592.805,E2 -9592.805} C_VEL
LIN {X 0,Y 432.205,Z 249.65,A -85,B 0,C 180,E1 -9594.394,E2 -9594.394} C_VEL
LIN {X 0,Y 432.21,Z 252.178,A -85,B 0,C 180,E1 -9596.436,E2 -9596.436} C_VEL
LIN {X 0,Y 432.081,Z 256.435,A -85,B 0,C 180,E1 -9599.72,E2 -9599.72} C_VEL
LIN {X 0,Y 431.854,Z 260.671,A -85,B 0,C 180,E1 -9602.892,E2 -9602.892} C_VEL
LIN {X 0,Y 431.783,Z 264.887,A -85,B 0,C 180,E1 -9605.989,E2 -9605.989} C_VEL
LIN {X 0,Y 431.597,Z 269.176,A -85,B 0,C 180,E1 -9609.008,E2 -9609.008} C_VEL
LIN {X 0,Y 431.502,Z 273.502,A -85,B 0,C 180,E1 -9611.973,E2 -9611.973} C_VEL
LIN {X 0,Y 431.514,Z 275.662,A -85,B 0,C 180,E1 -9613.38,E2 -9613.38} C_VEL
LIN {X 0,Y 434.411,Z 288.383,A -85,B 0,C 180,E1 -9613.889,E2 -9613.889} C_VEL
LIN {X 0,Y 435.928,Z 297.26,A -85,B 0,C 180,E1 -9614.333,E2 -9614.333} C_VEL
LIN {X 0,Y 435.367,Z 309.673,A -85,B 0,C 180,E1 -9615.032,E2 -9615.032} C_VEL
LIN {X 0,Y 434.746,Z 321.629,A -85,B 0,C 180,E1 -9615.918,E2 -9615.918} C_VEL
LIN {X 0,Y 434.123,Z 332.101,A -85,B 0,C 180,E1 -9616.9,E2 -9616.9} C_VEL
LIN {X 0,Y 433.441,Z 342.084,A -85,B 0,C 180,E1 -9618.069,E2 -9618.069} C_VEL
LIN {X 0,Y 432.773,Z 351.732,A -85,B 0,C 180,E1 -9619.473,E2 -9619.473} C_VEL
LIN {X 0,Y 432.245,Z 359.429,A -85,B 0,C 180,E1 -9620.879,E2 -9620.879} C_VEL
LIN {X 0,Y 431.799,Z 366.489,A -85,B 0,C 180,E1 -9622.518,E2 -9622.518} C_VEL
LIN {X 0,Y 431.622,Z 371.191,A -85,B 0,C 180,E1 -9623.925,E2 -9623.925} C_VEL
LIN {X 0,Y 431.355,Z 374.795,A -85,B 0,C 180,E1 -9625.327,E2 -9625.327} C_VEL
LIN {X 0,Y 431.309,Z 377.544,A -85,B 0,C 180,E1 -9626.857,E2 -9626.857} C_VEL
LIN {X 0,Y 430.64,Z 378.603,A -85,B 0,C 180,E1 -9627.625,E2 -9627.625} C_VEL
LIN {X 0,Y 427.714,Z 379.823,A -85,B 0,C 180,E1 -9628.881,E2 -9628.881} C_VEL
LIN {X 0,Y 425.236,Z 380.195,A -85,B 0,C 180,E1 -9629.9,E2 -9629.9} C_VEL
LIN {X 0,Y 424.175,Z 380.051,A -85,B 0,C 180,E1 -9630.688,E2 -9630.688} C_VEL
LIN {X 0,Y 424.091,Z 379.911,A -85,B 0,C 180,E1 -9630.955,E2 -9630.955} C_VEL
LIN {X 0,Y 424.237,Z 378.362,A -85,B 0,C 180,E1 -9632.849,E2 -9632.849} C_VEL
LIN {X 0,Y 424.223,Z 377.009,A -85,B 0,C 180,E1 -9633.8,E2 -9633.8} C_VEL
LIN {X 0,Y 424.375,Z 374.144,A -85,B 0,C 180,E1 -9635.226,E2 -9635.226} C_VEL
LIN {X 0,Y 424.634,Z 369.936,A -85,B 0,C 180,E1 -9636.76,E2 -9636.76} C_VEL
LIN {X 0,Y 424.844,Z 365.248,A -85,B 0,C 180,E1 -9638.083,E2 -9638.083} C_VEL
LIN {X 0,Y 425.316,Z 358.937,A -85,B 0,C 180,E1 -9639.511,E2 -9639.511} C_VEL
LIN {X 0,Y 425.883,Z 351.036,A -85,B 0,C 180,E1 -9640.94,E2 -9640.94} C_VEL
LIN {X 0,Y 426.434,Z 342.983,A -85,B 0,C 180,E1 -9642.13,E2 -9642.13} C_VEL
LIN {X 0,Y 427.179,Z 333.15,A -85,B 0,C 180,E1 -9643.317,E2 -9643.317} C_VEL
LIN {X 0,Y 427.816,Z 322.097,A -85,B 0,C 180,E1 -9644.387,E2 -9644.387} C_VEL
LIN {X 0,Y 428.461,Z 311.254,A -85,B 0,C 180,E1 -9645.215,E2 -9645.215} C_VEL
LIN {X 0,Y 429.045,Z 299.279,A -85,B 0,C 180,E1 -9645.925,E2 -9645.925} C_VEL
LIN {X 0,Y 427.967,Z 291.419,A -85,B 0,C 180,E1 -9646.342,E2 -9646.342} C_VEL
LIN {X 0,Y 425.103,Z 278.953,A -85,B 0,C 180,E1 -9646.892,E2 -9646.892} C_VEL
LIN {X 0,Y 424.423,Z 275.77,A -85,B 0,C 180,E1 -9647.023,E2 -9647.023} C_VEL
LIN {X 0,Y 424.507,Z 270.927,A -85,B 0,C 180,E1 -9650.345,E2 -9650.345} C_VEL
LIN {X 0,Y 424.637,Z 266.62,A -85,B 0,C 180,E1 -9653.404,E2 -9653.404} C_VEL
LIN {X 0,Y 424.814,Z 262.155,A -85,B 0,C 180,E1 -9656.701,E2 -9656.701} C_VEL
LIN {X 0,Y 424.948,Z 258.135,A -85,B 0,C 180,E1 -9659.746,E2 -9659.746} C_VEL
LIN {X 0,Y 425.101,Z 253.867,A -85,B 0,C 180,E1 -9663.064,E2 -9663.064} C_VEL
LIN {X 0,Y 425.173,Z 250.996,A -85,B 0,C 180,E1 -9665.348,E2 -9665.348} C_VEL
LIN {X 0,Y 425.163,Z 250.527,A -85,B 0,C 180,E1 -9665.906,E2 -9665.906} C_VEL
LIN {X 0,Y 425.283,Z 250.51,A -85,B 0,C 180,E1 -9668.901,E2 -9668.901} C_VEL
LIN {X 0,Y 425.259,Z 250.514,A -85,B 0,C 180,E1 -9672.655,E2 -9672.655} C_VEL
LIN {X 0,Y 425.286,Z 250.508,A -85,B 0,C 180,E1 -9675.283,E2 -9675.283} C_VEL
LIN {X 0,Y 425.27,Z 250.513,A -85,B 0,C 180,E1 -9678.621,E2 -9678.621} C_VEL
LIN {X 0,Y 425.296,Z 250.506,A -85,B 0,C 180,E1 -9681.101,E2 -9681.101} C_VEL
LIN {X 0,Y 425.301,Z 250.506,A -85,B 0,C 180,E1 -9684.664,E2 -9684.664} C_VEL
LIN {X 0,Y 425.267,Z 250.513,A -85,B 0,C 180,E1 -9688.073,E2 -9688.073} C_VEL
LIN {X 0,Y 425.333,Z 250.505,A -85,B 0,C 180,E1 -9691.368,E2 -9691.368} C_VEL
LIN {X 0,Y 425.357,Z 250.502,A -85,B 0,C 180,E1 -9693.505,E2 -9693.505} C_VEL
LIN {X 0,Y 425.288,Z 250.507,A -85,B 0,C 180,E1 -9696.634,E2 -9696.634} C_VEL
LIN {X 0,Y 425.298,Z 250.509,A -85,B 0,C 180,E1 -9699.695,E2 -9699.695} C_VEL
LIN {X 0,Y 425.333,Z 250.502,A -85,B 0,C 180,E1 -9702.697,E2 -9702.697} C_VEL
LIN {X 0,Y 425.347,Z 250.503,A -85,B 0,C 180,E1 -9705.65,E2 -9705.65} C_VEL
LIN {X 0,Y 425.355,Z 250.501,A -85,B 0,C 180,E1 -9708.564,E2 -9708.564} C_VEL
LIN {X 0,Y 425.508,Z 250.48,A -85,B 0,C 180,E1 -9712.31,E2 -9712.31} C_VEL
LIN {X 0,Y 425.543,Z 250.475,A -85,B 0,C 180,E1 -9714.313,E2 -9714.313} C_VEL
LIN {X 0,Y 425.57,Z 250.473,A -85,B 0,C 180,E1 -9718.107,E2 -9718.107} C_VEL
LIN {X 0,Y 425.523,Z 250.481,A -85,B 0,C 180,E1 -9720.946,E2 -9720.946} C_VEL
LIN {X 0,Y 425.549,Z 250.479,A -85,B 0,C 180,E1 -9722.84,E2 -9722.84} C_VEL
LIN {X 0,Y 425.551,Z 250.475,A -85,B 0,C 180,E1 -9725.687,E2 -9725.687} C_VEL
LIN {X 0,Y 425.407,Z 250.498,A -85,B 0,C 180,E1 -9728.551,E2 -9728.551} C_VEL
LIN {X 0,Y 425.411,Z 250.496,A -85,B 0,C 180,E1 -9732.402,E2 -9732.402} C_VEL
LIN {X 0,Y 425.392,Z 250.498,A -85,B 0,C 180,E1 -9736.312,E2 -9736.312} C_VEL
LIN {X 0,Y 425.332,Z 250.504,A -85,B 0,C 180,E1 -9739.636,E2 -9739.636} C_VEL
LIN {X 0,Y 425.29,Z 250.51,A -85,B 0,C 180,E1 -9742.339,E2 -9742.339} C_VEL
LIN {X 0,Y 425.263,Z 250.511,A -85,B 0,C 180,E1 -9745.447,E2 -9745.447} C_VEL
LIN {X 0,Y 425.315,Z 250.504,A -85,B 0,C 180,E1 -9748.861,E2 -9748.861} C_VEL
LIN {X 0,Y 425.267,Z 250.513,A -85,B 0,C 180,E1 -9751.927,E2 -9751.927} C_VEL
LIN {X 0,Y 425.301,Z 250.508,A -85,B 0,C 180,E1 -9755.336,E2 -9755.336} C_VEL
LIN {X 0,Y 425.282,Z 250.509,A -85,B 0,C 180,E1 -9758.901,E2 -9758.901} C_VEL
LIN {X 0,Y 425.262,Z 250.511,A -85,B 0,C 180,E1 -9762.655,E2 -9762.655} C_VEL
LIN {X 0,Y 425.287,Z 250.511,A -85,B 0,C 180,E1 -9765.283,E2 -9765.283} C_VEL
LIN {X 0,Y 425.28,Z 250.514,A -85,B 0,C 180,E1 -9768.622,E2 -9768.622} C_VEL
LIN {X 0,Y 425.333,Z 250.642,A -85,B 0,C 180,E1 -9769.679,E2 -9769.679} C_VEL
LIN {X 0,Y 426.123,Z 255.323,A -85,B 0,C 180,E1 -9772.393,E2 -9772.393} C_VEL
LIN {X 0,Y 426.487,Z 259.627,A -85,B 0,C 180,E1 -9774.777,E2 -9774.777} C_VEL
LIN {X 0,Y 426.177,Z 264.406,A -85,B 0,C 180,E1 -9777.249,E2 -9777.249} C_VEL
LIN {X 0,Y 425.777,Z 270.524,A -85,B 0,C 180,E1 -9780.318,E2 -9780.318} C_VEL
LIN {X 0,Y 425.377,Z 277.089,A -85,B 0,C 180,E1 -9783.507,E2 -9783.507} C_VEL
LIN {X 0,Y 425.08,Z 283.64,A -85,B 0,C 180,E1 -9786.621,E2 -9786.621} C_VEL
LIN {X 0,Y 424.799,Z 290.147,A -85,B 0,C 180,E1 -9789.67,E2 -9789.67} C_VEL
LIN {X 0,Y 424.579,Z 297.323,A -85,B 0,C 180,E1 -9793.018,E2 -9793.018} C_VEL
LIN {X 0,Y 426.94,Z 310.791,A -85,B 0,C 180,E1 -9793.513,E2 -9793.513} C_VEL
LIN {X 0,Y 428.614,Z 323.922,A -85,B 0,C 180,E1 -9794.181,E2 -9794.181} C_VEL
LIN {X 0,Y 427.932,Z 335.63,A -85,B 0,C 180,E1 -9794.887,E2 -9794.887} C_VEL
LIN {X 0,Y 427.172,Z 347.414,A -85,B 0,C 180,E1 -9795.815,E2 -9795.815} C_VEL
LIN {X 0,Y 426.455,Z 358.281,A -85,B 0,C 180,E1 -9796.903,E2 -9796.903} C_VEL
LIN {X 0,Y 425.927,Z 367.896,A -85,B 0,C 180,E1 -9798.097,E2 -9798.097} C_VEL
LIN {X 0,Y 425.278,Z 375.772,A -85,B 0,C 180,E1 -9799.285,E2 -9799.285} C_VEL
LIN {X 0,Y 424.82,Z 383.469,A -85,B 0,C 180,E1 -9800.718,E2 -9800.718} C_VEL
LIN {X 0,Y 424.436,Z 390.566,A -85,B 0,C 180,E1 -9802.388,E2 -9802.388} C_VEL
LIN {X 0,Y 424.243,Z 394.934,A -85,B 0,C 180,E1 -9803.7,E2 -9803.7} C_VEL
LIN {X 0,Y 424.2,Z 398.899,A -85,B 0,C 180,E1 -9805.248,E2 -9805.248} C_VEL
LIN {X 0,Y 424.098,Z 400.759,A -85,B 0,C 180,E1 -9806.199,E2 -9806.199} C_VEL
LIN {X 0,Y 424.131,Z 402.157,A -85,B 0,C 180,E1 -9807.15,E2 -9807.15} C_VEL
LIN {X 0,Y 424.129,Z 403.153,A -85,B 0,C 180,E1 -9808.101,E2 -9808.101} C_VEL
LIN {X 0,Y 424.084,Z 403.976,A -85,B 0,C 180,E1 -9810,E2 -9810} C_VEL
LIN {X 0,Y 424.129,Z 403.152,A -85,B 0,C 180,E1 -9811.899,E2 -9811.899} C_VEL
LIN {X 0,Y 424.131,Z 402.156,A -85,B 0,C 180,E1 -9812.849,E2 -9812.849} C_VEL
LIN {X 0,Y 424.098,Z 400.757,A -85,B 0,C 180,E1 -9813.801,E2 -9813.801} C_VEL
LIN {X 0,Y 424.207,Z 397.82,A -85,B 0,C 180,E1 -9815.228,E2 -9815.228} C_VEL
LIN {X 0,Y 424.301,Z 393.843,A -85,B 0,C 180,E1 -9816.658,E2 -9816.658} C_VEL
LIN {X 0,Y 424.588,Z 387.73,A -85,B 0,C 180,E1 -9818.328,E2 -9818.328} C_VEL
LIN {X 0,Y 424.956,Z 381.05,A -85,B 0,C 180,E1 -9819.76,E2 -9819.76} C_VEL
LIN {X 0,Y 425.481,Z 372.764,A -85,B 0,C 180,E1 -9821.191,E2 -9821.191} C_VEL
LIN {X 0,Y 426.149,Z 364.275,A -85,B 0,C 180,E1 -9822.38,E2 -9822.38} C_VEL
LIN {X 0,Y 426.766,Z 354.28,A -85,B 0,C 180,E1 -9823.521,E2 -9823.521} C_VEL
LIN {X 0,Y 427.446,Z 343.401,A -85,B 0,C 180,E1 -9824.521,E2 -9824.521} C_VEL
LIN {X 0,Y 428.161,Z 332.024,A -85,B 0,C 180,E1 -9825.348,E2 -9825.348} C_VEL
LIN {X 0,Y 428.48,Z 322.688,A -85,B 0,C 180,E1 -9825.885,E2 -9825.885} C_VEL
LIN {X 0,Y 426.731,Z 309.579,A -85,B 0,C 180,E1 -9826.535,E2 -9826.535} C_VEL
LIN {X 0,Y 424.585,Z 297.282,A -85,B 0,C 180,E1 -9826.996,E2 -9826.996} C_VEL
LIN {X 0,Y 424.862,Z 289.042,A -85,B 0,C 180,E1 -9830.833,E2 -9830.833} C_VEL
LIN {X 0,Y 425.126,Z 282.538,A -85,B 0,C 180,E1 -9833.893,E2 -9833.893} C_VEL
LIN {X 0,Y 425.396,Z 276.299,A -85,B 0,C 180,E1 -9836.856,E2 -9836.856} C_VEL
LIN {X 0,Y 425.844,Z 269.386,A -85,B 0,C 180,E1 -9840.223,E2 -9840.223} C_VEL
LIN {X 0,Y 426.298,Z 262.866,A -85,B 0,C 180,E1 -9843.524,E2 -9843.524} C_VEL
LIN {X 0,Y 426.488,Z 259.62,A -85,B 0,C 180,E1 -9845.223,E2 -9845.223} C_VEL
LIN {X 0,Y 426.092,Z 255.208,A -85,B 0,C 180,E1 -9847.654,E2 -9847.654} C_VEL
LIN {X 0,Y 425.314,Z 250.511,A -85,B 0,C 180,E1 -9850.446,E2 -9850.446} C_VEL
LIN {X 0,Y 425.263,Z 250.514,A -85,B 0,C 180,E1 -9853.956,E2 -9853.956} C_VEL
LIN {X 0,Y 425.25,Z 250.515,A -85,B 0,C 180,E1 -9856.65,E2 -9856.65} C_VEL
LIN {X 0,Y 425.245,Z 250.512,A -85,B 0,C 180,E1 -9859.868,E2 -9859.868} C_VEL
LIN {X 0,Y 425.276,Z 250.514,A -85,B 0,C 180,E1 -9862.489,E2 -9862.489} C_VEL
LIN {X 0,Y 425.308,Z 250.507,A -85,B 0,C 180,E1 -9865.817,E2 -9865.817} C_VEL
LIN {X 0,Y 425.292,Z 250.508,A -85,B 0,C 180,E1 -9869.239,E2 -9869.239} C_VEL
LIN {X 0,Y 425.27,Z 250.513,A -85,B 0,C 180,E1 -9872.437,E2 -9872.437} C_VEL
LIN {X 0,Y 425.324,Z 250.504,A -85,B 0,C 180,E1 -9875.6,E2 -9875.6} C_VEL
LIN {X 0,Y 425.295,Z 250.507,A -85,B 0,C 180,E1 -9878.682,E2 -9878.682} C_VEL
LIN {X 0,Y 425.335,Z 250.505,A -85,B 0,C 180,E1 -9881.703,E2 -9881.703} C_VEL
LIN {X 0,Y 425.349,Z 250.5,A -85,B 0,C 180,E1 -9884.671,E2 -9884.671} C_VEL
LIN {X 0,Y 425.413,Z 250.495,A -85,B 0,C 180,E1 -9887.598,E2 -9887.598} C_VEL
LIN {X 0,Y 425.409,Z 250.497,A -85,B 0,C 180,E1 -9891.449,E2 -9891.449} C_VEL
LIN {X 0,Y 425.55,Z 250.475,A -85,B 0,C 180,E1 -9894.313,E2 -9894.313} C_VEL
LIN {X 0,Y 425.574,Z 250.473,A -85,B 0,C 180,E1 -9898.107,E2 -9898.107} C_VEL
LIN {X 0,Y 425.699,Z 250.457,A -85,B 0,C 180,E1 -9900,E2 -9900} C_VEL
LIN {X 0,Y 425.523,Z 250.48,A -85,B 0,C 180,E1 -9902.84,E2 -9902.84} C_VEL
LIN {X 0,Y 425.542,Z 250.475,A -85,B 0,C 180,E1 -9905.687,E2 -9905.687} C_VEL
LIN {X 0,Y 425.41,Z 250.495,A -85,B 0,C 180,E1 -9908.551,E2 -9908.551} C_VEL
LIN {X 0,Y 425.414,Z 250.495,A -85,B 0,C 180,E1 -9912.402,E2 -9912.402} C_VEL
LIN {X 0,Y 425.389,Z 250.497,A -85,B 0,C 180,E1 -9916.312,E2 -9916.312} C_VEL
LIN {X 0,Y 425.33,Z 250.501,A -85,B 0,C 180,E1 -9919.635,E2 -9919.635} C_VEL
LIN {X 0,Y 425.29,Z 250.512,A -85,B 0,C 180,E1 -9922.339,E2 -9922.339} C_VEL
LIN {X 0,Y 425.292,Z 250.507,A -85,B 0,C 180,E1 -9925.446,E2 -9925.446} C_VEL
LIN {X 0,Y 425.35,Z 250.501,A -85,B 0,C 180,E1 -9927.558,E2 -9927.558} C_VEL
LIN {X 0,Y 425.289,Z 250.509,A -85,B 0,C 180,E1 -9930.816,E2 -9930.816} C_VEL
LIN {X 0,Y 425.292,Z 250.51,A -85,B 0,C 180,E1 -9934.284,E2 -9934.284} C_VEL
LIN {X 0,Y 425.278,Z 250.512,A -85,B 0,C 180,E1 -9937.695,E2 -9937.695} C_VEL
LIN {X 0,Y 425.278,Z 250.51,A -85,B 0,C 180,E1 -9940.52,E2 -9940.52} C_VEL
LIN {X 0,Y 425.261,Z 250.515,A -85,B 0,C 180,E1 -9943.956,E2 -9943.956} C_VEL
LIN {X 0,Y 425.245,Z 250.513,A -85,B 0,C 180,E1 -9946.651,E2 -9946.651} C_VEL
LIN {X 0,Y 425.244,Z 250.515,A -85,B 0,C 180,E1 -9949.868,E2 -9949.868} C_VEL
LIN {X 0,Y 425.272,Z 250.511,A -85,B 0,C 180,E1 -9952.49,E2 -9952.49} C_VEL
LIN {X 0,Y 425.167,Z 250.526,A -85,B 0,C 180,E1 -9954.093,E2 -9954.093} C_VEL
LIN {X 0,Y 425.18,Z 250.869,A -85,B 0,C 180,E1 -9954.653,E2 -9954.653} C_VEL
LIN {X 0,Y 425.115,Z 254.403,A -85,B 0,C 180,E1 -9957.473,E2 -9957.473} C_VEL
LIN {X 0,Y 424.958,Z 257.992,A -85,B 0,C 180,E1 -9960.255,E2 -9960.255} C_VEL
LIN {X 0,Y 424.806,Z 262.231,A -85,B 0,C 180,E1 -9963.469,E2 -9963.469} C_VEL
LIN {X 0,Y 424.639,Z 266.478,A -85,B 0,C 180,E1 -9966.596,E2 -9966.596} C_VEL
LIN {X 0,Y 424.505,Z 270.783,A -85,B 0,C 180,E1 -9969.655,E2 -9969.655} C_VEL
LIN {X 0,Y 424.446,Z 275.936,A -85,B 0,C 180,E1 -9973.096,E2 -9973.096} C_VEL
LIN {X 0,Y 427.517,Z 289.277,A -85,B 0,C 180,E1 -9973.649,E2 -9973.649} C_VEL
LIN {X 0,Y 429.076,Z 298.639,A -85,B 0,C 180,E1 -9974.137,E2 -9974.137} C_VEL
LIN {X 0,Y 428.505,Z 309.88,A -85,B 0,C 180,E1 -9974.786,E2 -9974.786} C_VEL
LIN {X 0,Y 427.911,Z 320.987,A -85,B 0,C 180,E1 -9975.616,E2 -9975.616} C_VEL
LIN {X 0,Y 427.211,Z 332.305,A -85,B 0,C 180,E1 -9976.685,E2 -9976.685} C_VEL
LIN {X 0,Y 426.501,Z 342.287,A -85,B 0,C 180,E1 -9977.872,E2 -9977.872} C_VEL
LIN {X 0,Y 425.797,Z 351.934,A -85,B 0,C 180,E1 -9979.299,E2 -9979.299} C_VEL
LIN {X 0,Y 425.229,Z 359.631,A -85,B 0,C 180,E1 -9980.727,E2 -9980.727} C_VEL
LIN {X 0,Y 424.751,Z 366.691,A -85,B 0,C 180,E1 -9982.394,E2 -9982.394} C_VEL
LIN {X 0,Y 424.574,Z 370.791,A -85,B 0,C 180,E1 -9983.621,E2 -9983.621} C_VEL
LIN {X 0,Y 424.288,Z 374.995,A -85,B 0,C 180,E1 -9985.249,E2 -9985.249} C_VEL
LIN {X 0,Y 424.222,Z 377.818,A -85,B 0,C 180,E1 -9986.855,E2 -9986.855} C_VEL
LIN {X 0,Y 424.152,Z 379.253,A -85,B 0,C 180,E1 -9988.101,E2 -9988.101} C_VEL
LIN {X 0,Y 424.085,Z 380.102,A -85,B 0,C 180,E1 -9990,E2 -9990} C_VEL
LIN {X 0,Y 424.091,Z 379.911,A -85,B 0,C 180,E1 -9990.955,E2 -9990.955} C_VEL
LIN {X 0,Y 423.426,Z 379.481,A -85,B 0,C 180,E1 -9991.746,E2 -9991.746} C_VEL
LIN {X 0,Y 420.578,Z 378.288,A -85,B 0,C 180,E1 -9993.026,E2 -9993.026} C_VEL
LIN {X 0,Y 418.227,Z 376.842,A -85,B 0,C 180,E1 -9994.05,E2 -9994.05} C_VEL
LIN {X 0,Y 417.302,Z 375.401,A -85,B 0,C 180,E1 -9994.829,E2 -9994.829} C_VEL
LIN {X 0,Y 417.271,Z 374.834,A -85,B 0,C 180,E1 -9995.09,E2 -9995.09} C_VEL
LIN {X 0,Y 417.562,Z 370.457,A -85,B 0,C 180,E1 -9996.766,E2 -9996.766} C_VEL
LIN {X 0,Y 417.808,Z 365.447,A -85,B 0,C 180,E1 -9998.22,E2 -9998.22} C_VEL
LIN {X 0,Y 418.315,Z 359.135,A -85,B 0,C 180,E1 -9999.672,E2 -9999.672} C_VEL
LIN {X 0,Y 418.918,Z 351.233,A -85,B 0,C 180,E1 -10001.124,E2 -10001.124} C_VEL
LIN {X 0,Y 419.476,Z 343.18,A -85,B 0,C 180,E1 -10002.335,E2 -10002.335} C_VEL
LIN {X 0,Y 420.279,Z 333.346,A -85,B 0,C 180,E1 -10003.539,E2 -10003.539} C_VEL
LIN {X 0,Y 420.94,Z 322.291,A -85,B 0,C 180,E1 -10004.627,E2 -10004.627} C_VEL
LIN {X 0,Y 421.61,Z 311.447,A -85,B 0,C 180,E1 -10005.469,E2 -10005.469} C_VEL
LIN {X 0,Y 422.223,Z 299.559,A -85,B 0,C 180,E1 -10006.184,E2 -10006.184} C_VEL
LIN {X 0,Y 420.315,Z 288.454,A -85,B 0,C 180,E1 -10006.779,E2 -10006.779} C_VEL
LIN {X 0,Y 417.344,Z 275.966,A -85,B 0,C 180,E1 -10007.324,E2 -10007.324} C_VEL
LIN {X 0,Y 417.449,Z 272.541,A -85,B 0,C 180,E1 -10009.677,E2 -10009.677} C_VEL
LIN {X 0,Y 417.527,Z 268.226,A -85,B 0,C 180,E1 -10012.777,E2 -10012.777} C_VEL
LIN {X 0,Y 417.704,Z 263.934,A -85,B 0,C 180,E1 -10015.942,E2 -10015.942} C_VEL
LIN {X 0,Y 417.869,Z 259.695,A -85,B 0,C 180,E1 -10019.192,E2 -10019.192} C_VEL
LIN {X 0,Y 418.045,Z 255.423,A -85,B 0,C 180,E1 -10022.546,E2 -10022.546} C_VEL
LIN {X 0,Y 418.119,Z 252.546,A -85,B 0,C 180,E1 -10024.855,E2 -10024.855} C_VEL
LIN {X 0,Y 418.162,Z 251.399,A -85,B 0,C 180,E1 -10026.222,E2 -10026.222} C_VEL
LIN {X 0,Y 418.21,Z 251.388,A -85,B 0,C 180,E1 -10029.373,E2 -10029.373} C_VEL
LIN {X 0,Y 418.211,Z 251.394,A -85,B 0,C 180,E1 -10032.318,E2 -10032.318} C_VEL
LIN {X 0,Y 418.237,Z 251.387,A -85,B 0,C 180,E1 -10035.109,E2 -10035.109} C_VEL
LIN {X 0,Y 418.236,Z 251.388,A -85,B 0,C 180,E1 -10037.766,E2 -10037.766} C_VEL
LIN {X 0,Y 418.246,Z 251.387,A -85,B 0,C 180,E1 -10040.621,E2 -10040.621} C_VEL
LIN {X 0,Y 418.245,Z 251.389,A -85,B 0,C 180,E1 -10043.976,E2 -10043.976} C_VEL
LIN {X 0,Y 418.26,Z 251.383,A -85,B 0,C 180,E1 -10047.156,E2 -10047.156} C_VEL
LIN {X 0,Y 418.271,Z 251.382,A -85,B 0,C 180,E1 -10050.896,E2 -10050.896} C_VEL
LIN {X 0,Y 418.271,Z 251.384,A -85,B 0,C 180,E1 -10054.096,E2 -10054.096} C_VEL
LIN {X 0,Y 418.235,Z 251.388,A -85,B 0,C 180,E1 -10057.264,E2 -10057.264} C_VEL
LIN {X 0,Y 418.286,Z 251.379,A -85,B 0,C 180,E1 -10060.364,E2 -10060.364} C_VEL
LIN {X 0,Y 418.318,Z 251.379,A -85,B 0,C 180,E1 -10063.405,E2 -10063.405} C_VEL
LIN {X 0,Y 418.35,Z 251.375,A -85,B 0,C 180,E1 -10066.999,E2 -10066.999} C_VEL
LIN {X 0,Y 418.343,Z 251.373,A -85,B 0,C 180,E1 -10070.329,E2 -10070.329} C_VEL
LIN {X 0,Y 418.471,Z 251.36,A -85,B 0,C 180,E1 -10073.249,E2 -10073.249} C_VEL
LIN {X 0,Y 418.327,Z 251.377,A -85,B 0,C 180,E1 -10075.181,E2 -10075.181} C_VEL
LIN {X 0,Y 418.539,Z 251.348,A -85,B 0,C 180,E1 -10078.075,E2 -10078.075} C_VEL
LIN {X 0,Y 418.485,Z 251.358,A -85,B 0,C 180,E1 -10080.962,E2 -10080.962} C_VEL
LIN {X 0,Y 418.504,Z 251.356,A -85,B 0,C 180,E1 -10082.888,E2 -10082.888} C_VEL
LIN {X 0,Y 418.509,Z 251.352,A -85,B 0,C 180,E1 -10085.783,E2 -10085.783} C_VEL
LIN {X 0,Y 418.376,Z 251.372,A -85,B 0,C 180,E1 -10088.696,E2 -10088.696} C_VEL
LIN {X 0,Y 418.356,Z 251.374,A -85,B 0,C 180,E1 -10092.614,E2 -10092.614} C_VEL
LIN {X 0,Y 418.304,Z 251.378,A -85,B 0,C 180,E1 -10095.594,E2 -10095.594} C_VEL
LIN {X 0,Y 418.287,Z 251.382,A -85,B 0,C 180,E1 -10098.617,E2 -10098.617} C_VEL
LIN {X 0,Y 418.237,Z 251.388,A -85,B 0,C 180,E1 -10101.696,E2 -10101.696} C_VEL
LIN {X 0,Y 418.246,Z 251.383,A -85,B 0,C 180,E1 -10104.852,E2 -10104.852} C_VEL
LIN {X 0,Y 418.247,Z 251.387,A -85,B 0,C 180,E1 -10108.067,E2 -10108.067} C_VEL
LIN {X 0,Y 418.214,Z 251.392,A -85,B 0,C 180,E1 -10111.396,E2 -10111.396} C_VEL
LIN {X 0,Y 418.268,Z 251.382,A -85,B 0,C 180,E1 -10114.58,E2 -10114.58} C_VEL
LIN {X 0,Y 418.223,Z 251.39,A -85,B 0,C 180,E1 -10117.832,E2 -10117.832} C_VEL
LIN {X 0,Y 418.21,Z 251.39,A -85,B 0,C 180,E1 -10120.95,E2 -10120.95} C_VEL
LIN {X 0,Y 418.206,Z 251.392,A -85,B 0,C 180,E1 -10123.728,E2 -10123.728} C_VEL
LIN {X 0,Y 418.211,Z 251.393,A -85,B 0,C 180,E1 -10126.449,E2 -10126.449} C_VEL
LIN {X 0,Y 418.281,Z 251.516,A -85,B 0,C 180,E1 -10129.427,E2 -10129.427} C_VEL
LIN {X 0,Y 419.041,Z 255.883,A -85,B 0,C 180,E1 -10132.024,E2 -10132.024} C_VEL
LIN {X 0,Y 419.497,Z 260.617,A -85,B 0,C 180,E1 -10134.691,E2 -10134.691} C_VEL
LIN {X 0,Y 419.097,Z 266.029,A -85,B 0,C 180,E1 -10137.546,E2 -10137.546} C_VEL
LIN {X 0,Y 418.655,Z 272.562,A -85,B 0,C 180,E1 -10140.868,E2 -10140.868} C_VEL
LIN {X 0,Y 418.225,Z 280.218,A -85,B 0,C 180,E1 -10144.627,E2 -10144.627} C_VEL
LIN {X 0,Y 417.882,Z 287.809,A -85,B 0,C 180,E1 -10148.284,E2 -10148.284} C_VEL
LIN {X 0,Y 417.528,Z 295.314,A -85,B 0,C 180,E1 -10151.856,E2 -10151.856} C_VEL
LIN {X 0,Y 417.525,Z 297.094,A -85,B 0,C 180,E1 -10152.704,E2 -10152.704} C_VEL
LIN {X 0,Y 420.196,Z 312.364,A -85,B 0,C 180,E1 -10153.313,E2 -10153.313} C_VEL
LIN {X 0,Y 421.72,Z 324.859,A -85,B 0,C 180,E1 -10153.977,E2 -10153.977} C_VEL
LIN {X 0,Y 420.944,Z 337.12,A -85,B 0,C 180,E1 -10154.754,E2 -10154.754} C_VEL
LIN {X 0,Y 420.149,Z 348.779,A -85,B 0,C 180,E1 -10155.722,E2 -10155.722} C_VEL
LIN {X 0,Y 419.436,Z 359.156,A -85,B 0,C 180,E1 -10156.803,E2 -10156.803} C_VEL
LIN {X 0,Y 418.938,Z 367.697,A -85,B 0,C 180,E1 -10157.895,E2 -10157.895} C_VEL
LIN {X 0,Y 418.28,Z 375.573,A -85,B 0,C 180,E1 -10159.104,E2 -10159.104} C_VEL
LIN {X 0,Y 417.784,Z 383.269,A -85,B 0,C 180,E1 -10160.56,E2 -10160.56} C_VEL
LIN {X 0,Y 417.37,Z 390.367,A -85,B 0,C 180,E1 -10162.258,E2 -10162.258} C_VEL
LIN {X 0,Y 417.167,Z 395.07,A -85,B 0,C 180,E1 -10163.707,E2 -10163.707} C_VEL
LIN {X 0,Y 417.107,Z 398.7,A -85,B 0,C 180,E1 -10165.167,E2 -10165.167} C_VEL
LIN {X 0,Y 417.014,Z 400.56,A -85,B 0,C 180,E1 -10166.134,E2 -10166.134} C_VEL
LIN {X 0,Y 417.028,Z 401.957,A -85,B 0,C 180,E1 -10167.102,E2 -10167.102} C_VEL
LIN {X 0,Y 417.056,Z 402.954,A -85,B 0,C 180,E1 -10168.068,E2 -10168.068} C_VEL
LIN {X 0,Y 417.004,Z 403.777,A -85,B 0,C 180,E1 -10170,E2 -10170} C_VEL
LIN {X 0,Y 417.056,Z 402.953,A -85,B 0,C 180,E1 -10171.931,E2 -10171.931} C_VEL
LIN {X 0,Y 417.028,Z 401.955,A -85,B 0,C 180,E1 -10172.898,E2 -10172.898} C_VEL
LIN {X 0,Y 417.014,Z 400.556,A -85,B 0,C 180,E1 -10173.865,E2 -10173.865} C_VEL
LIN {X 0,Y 417.122,Z 397.619,A -85,B 0,C 180,E1 -10175.317,E2 -10175.317} C_VEL
LIN {X 0,Y 417.234,Z 393.642,A -85,B 0,C 180,E1 -10176.771,E2 -10176.771} C_VEL
LIN {X 0,Y 417.528,Z 387.527,A -85,B 0,C 180,E1 -10178.469,E2 -10178.469} C_VEL
LIN {X 0,Y 417.934,Z 380.848,A -85,B 0,C 180,E1 -10179.925,E2 -10179.925} C_VEL
LIN {X 0,Y 418.503,Z 372.562,A -85,B 0,C 180,E1 -10181.38,E2 -10181.38} C_VEL
LIN {X 0,Y 419.178,Z 364.071,A -85,B 0,C 180,E1 -10182.589,E2 -10182.589} C_VEL
LIN {X 0,Y 419.827,Z 353.908,A -85,B 0,C 180,E1 -10183.766,E2 -10183.766} C_VEL
LIN {X 0,Y 420.539,Z 343.197,A -85,B 0,C 180,E1 -10184.765,E2 -10184.765} C_VEL
LIN {X 0,Y 421.327,Z 331.819,A -85,B 0,C 180,E1 -10185.603,E2 -10185.603} C_VEL
LIN {X 0,Y 421.61,Z 323.614,A -85,B 0,C 180,E1 -10186.089,E2 -10186.089} C_VEL
LIN {X 0,Y 419.913,Z 310.745,A -85,B 0,C 180,E1 -10186.758,E2 -10186.758} C_VEL
LIN {X 0,Y 417.589,Z 297.875,A -85,B 0,C 180,E1 -10187.252,E2 -10187.252} C_VEL
LIN {X 0,Y 417.527,Z 297.075,A -85,B 0,C 180,E1 -10187.296,E2 -10187.296} C_VEL
LIN {X 0,Y 417.831,Z 288.867,A -85,B 0,C 180,E1 -10191.201,E2 -10191.201} C_VEL
LIN {X 0,Y 418.195,Z 281.298,A -85,B 0,C 180,E1 -10194.843,E2 -10194.843} C_VEL
LIN {X 0,Y 418.586,Z 273.616,A -85,B 0,C 180,E1 -10198.588,E2 -10198.588} C_VEL
LIN {X 0,Y 419.025,Z 267.089,A -85,B 0,C 180,E1 -10201.892,E2 -10201.892} C_VEL
LIN {X 0,Y 419.431,Z 261.522,A -85,B 0,C 180,E1 -10204.81,E2 -10204.81} C_VEL
LIN {X 0,Y 419.236,Z 257.342,A -85,B 0,C 180,E1 -10207.121,E2 -10207.121} C_VEL
LIN {X 0,Y 418.38,Z 252.004,A -85,B 0,C 180,E1 -10210.262,E2 -10210.262} C_VEL
LIN {X 0,Y 418.247,Z 251.394,A -85,B 0,C 180,E1 -10210.793,E2 -10210.793} C_VEL
LIN {X 0,Y 418.211,Z 251.394,A -85,B 0,C 180,E1 -10213.729,E2 -10213.729} C_VEL
LIN {X 0,Y 418.203,Z 251.393,A -85,B 0,C 180,E1 -10216.448,E2 -10216.448} C_VEL
LIN {X 0,Y 418.209,Z 251.39,A -85,B 0,C 180,E1 -10219.133,E2 -10219.133} C_VEL
LIN {X 0,Y 418.239,Z 251.388,A -85,B 0,C 180,E1 -10222.776,E2 -10222.776} C_VEL
LIN {X 0,Y 418.25,Z 251.388,A -85,B 0,C 180,E1 -10226.323,E2 -10226.323} C_VEL
LIN {X 0,Y 418.243,Z 251.387,A -85,B 0,C 180,E1 -10229.728,E2 -10229.728} C_VEL
LIN {X 0,Y 418.227,Z 251.387,A -85,B 0,C 180,E1 -10233.018,E2 -10233.018} C_VEL
LIN {X 0,Y 418.26,Z 251.386,A -85,B 0,C 180,E1 -10236.217,E2 -10236.217} C_VEL
LIN {X 0,Y 418.252,Z 251.385,A -85,B 0,C 180,E1 -10239.337,E2 -10239.337} C_VEL
LIN {X 0,Y 418.29,Z 251.381,A -85,B 0,C 180,E1 -10242.396,E2 -10242.396} C_VEL
LIN {X 0,Y 418.303,Z 251.38,A -85,B 0,C 180,E1 -10245.403,E2 -10245.403} C_VEL
LIN {X 0,Y 418.313,Z 251.376,A -85,B 0,C 180,E1 -10248.369,E2 -10248.369} C_VEL
LIN {X 0,Y 418.467,Z 251.357,A -85,B 0,C 180,E1 -10252.279,E2 -10252.279} C_VEL
LIN {X 0,Y 418.508,Z 251.352,A -85,B 0,C 180,E1 -10254.217,E2 -10254.217} C_VEL
LIN {X 0,Y 418.544,Z 251.348,A -85,B 0,C 180,E1 -10258.076,E2 -10258.076} C_VEL
LIN {X 0,Y 418.668,Z 251.333,A -85,B 0,C 180,E1 -10260,E2 -10260} C_VEL
LIN {X 0,Y 418.48,Z 251.358,A -85,B 0,C 180,E1 -10262.888,E2 -10262.888} C_VEL
LIN {X 0,Y 418.467,Z 251.359,A -85,B 0,C 180,E1 -10266.628,E2 -10266.628} C_VEL
LIN {X 0,Y 418.342,Z 251.373,A -85,B 0,C 180,E1 -10269.671,E2 -10269.671} C_VEL
LIN {X 0,Y 418.348,Z 251.375,A -85,B 0,C 180,E1 -10273.001,E2 -10273.001} C_VEL
LIN {X 0,Y 418.314,Z 251.38,A -85,B 0,C 180,E1 -10276.735,E2 -10276.735} C_VEL
LIN {X 0,Y 418.272,Z 251.381,A -85,B 0,C 180,E1 -10279.79,E2 -10279.79} C_VEL
LIN {X 0,Y 418.233,Z 251.388,A -85,B 0,C 180,E1 -10282.737,E2 -10282.737} C_VEL
LIN {X 0,Y 418.27,Z 251.384,A -85,B 0,C 180,E1 -10285.904,E2 -10285.904} C_VEL
LIN {X 0,Y 418.266,Z 251.382,A -85,B 0,C 180,E1 -10289.162,E2 -10289.162} C_VEL
LIN {X 0,Y 418.252,Z 251.384,A -85,B 0,C 180,E1 -10292.843,E2 -10292.843} C_VEL
LIN {X 0,Y 418.245,Z 251.387,A -85,B 0,C 180,E1 -10296.238,E2 -10296.238} C_VEL
LIN {X 0,Y 418.243,Z 251.389,A -85,B 0,C 180,E1 -10299.683,E2 -10299.683} C_VEL
LIN {X 0,Y 418.225,Z 251.389,A -85,B 0,C 180,E1 -10302.32,E2 -10302.32} C_VEL
LIN {X 0,Y 418.235,Z 251.388,A -85,B 0,C 180,E1 -10305.108,E2 -10305.108} C_VEL
LIN {X 0,Y 418.219,Z 251.393,A -85,B 0,C 180,E1 -10307.764,E2 -10307.764} C_VEL
LIN {X 0,Y 418.238,Z 251.39,A -85,B 0,C 180,E1 -10311.557,E2 -10311.557} C_VEL
LIN {X 0,Y 418.149,Z 251.4,A -85,B 0,C 180,E1 -10313.966,E2 -10313.966} C_VEL
LIN {X 0,Y 418.136,Z 252.779,A -85,B 0,C 180,E1 -10315.446,E2 -10315.446} C_VEL
LIN {X 0,Y 417.991,Z 256.708,A -85,B 0,C 180,E1 -10318.585,E2 -10318.585} C_VEL
LIN {X 0,Y 417.809,Z 260.97,A -85,B 0,C 180,E1 -10321.901,E2 -10321.901} C_VEL
LIN {X 0,Y 417.65,Z 265.481,A -85,B 0,C 180,E1 -10325.325,E2 -10325.325} C_VEL
LIN {X 0,Y 417.511,Z 269.524,A -85,B 0,C 180,E1 -10328.264,E2 -10328.264} C_VEL
LIN {X 0,Y 417.39,Z 273.877,A -85,B 0,C 180,E1 -10331.342,E2 -10331.342} C_VEL
LIN {X 0,Y 417.377,Z 276.081,A -85,B 0,C 180,E1 -10332.799,E2 -10332.799} C_VEL
LIN {X 0,Y 420.403,Z 289.014,A -85,B 0,C 180,E1 -10333.345,E2 -10333.345} C_VEL
LIN {X 0,Y 422.206,Z 299.635,A -85,B 0,C 180,E1 -10333.916,E2 -10333.916} C_VEL
LIN {X 0,Y 421.592,Z 311.848,A -85,B 0,C 180,E1 -10334.655,E2 -10334.655} C_VEL
LIN {X 0,Y 420.928,Z 323.307,A -85,B 0,C 180,E1 -10335.557,E2 -10335.557} C_VEL
LIN {X 0,Y 420.223,Z 333.585,A -85,B 0,C 180,E1 -10336.582,E2 -10336.582} C_VEL
LIN {X 0,Y 419.555,Z 342.49,A -85,B 0,C 180,E1 -10337.668,E2 -10337.668} C_VEL
LIN {X 0,Y 418.831,Z 352.137,A -85,B 0,C 180,E1 -10339.119,E2 -10339.119} C_VEL
LIN {X 0,Y 418.217,Z 359.833,A -85,B 0,C 180,E1 -10340.57,E2 -10340.57} C_VEL
LIN {X 0,Y 417.7,Z 366.893,A -85,B 0,C 180,E1 -10342.264,E2 -10342.264} C_VEL
LIN {X 0,Y 417.487,Z 371.28,A -85,B 0,C 180,E1 -10343.61,E2 -10343.61} C_VEL
LIN {X 0,Y 417.226,Z 375.196,A -85,B 0,C 180,E1 -10345.169,E2 -10345.169} C_VEL
LIN {X 0,Y 417.135,Z 377.056,A -85,B 0,C 180,E1 -10346.136,E2 -10346.136} C_VEL
LIN {X 0,Y 417.154,Z 378.455,A -85,B 0,C 180,E1 -10347.103,E2 -10347.103} C_VEL
LIN {X 0,Y 417.014,Z 380.068,A -85,B 0,C 180,E1 -10349.034,E2 -10349.034} C_VEL
LIN {X 0,Y 417.004,Z 380.302,A -85,B 0,C 180,E1 -10350,E2 -10350} C_VEL
LIN {X 0,Y 417.014,Z 380.114,A -85,B 0,C 180,E1 -10350.966,E2 -10350.966} C_VEL
LIN {X 0,Y 417.153,Z 378.562,A -85,B 0,C 180,E1 -10352.897,E2 -10352.897} C_VEL
LIN {X 0,Y 417.131,Z 377.209,A -85,B 0,C 180,E1 -10353.864,E2 -10353.864} C_VEL
LIN {X 0,Y 417.271,Z 374.834,A -85,B 0,C 180,E1 -10355.09,E2 -10355.09} C_VEL
LIN {X 0,Y 416.75,Z 373.053,A -85,B 0,C 180,E1 -10355.86,E2 -10355.86} C_VEL
LIN {X 0,Y 414.08,Z 369.719,A -85,B 0,C 180,E1 -10357.094,E2 -10357.094} C_VEL
LIN {X 0,Y 411.439,Z 365.778,A -85,B 0,C 180,E1 -10358.307,E2 -10358.307} C_VEL
LIN {X 0,Y 410.979,Z 362.945,A -85,B 0,C 180,E1 -10359.033,E2 -10359.033} C_VEL
LIN {X 0,Y 411.564,Z 355.598,A -85,B 0,C 180,E1 -10360.578,E2 -10360.578} C_VEL
LIN {X 0,Y 412.293,Z 346.786,A -85,B 0,C 180,E1 -10362.053,E2 -10362.053} C_VEL
LIN {X 0,Y 413.052,Z 337.742,A -85,B 0,C 180,E1 -10363.28,E2 -10363.28} C_VEL
LIN {X 0,Y 413.79,Z 327.456,A -85,B 0,C 180,E1 -10364.41,E2 -10364.41} C_VEL
LIN {X 0,Y 414.467,Z 316.591,A -85,B 0,C 180,E1 -10365.364,E2 -10365.364} C_VEL
LIN {X 0,Y 415.209,Z 304.586,A -85,B 0,C 180,E1 -10366.186,E2 -10366.186} C_VEL
LIN {X 0,Y 415.302,Z 299.464,A -85,B 0,C 180,E1 -10366.478,E2 -10366.478} C_VEL
LIN {X 0,Y 412.997,Z 287.471,A -85,B 0,C 180,E1 -10367.134,E2 -10367.134} C_VEL
LIN {X 0,Y 410.273,Z 276.168,A -85,B 0,C 180,E1 -10367.625,E2 -10367.625} C_VEL
LIN {X 0,Y 410.371,Z 272.725,A -85,B 0,C 180,E1 -10370.031,E2 -10370.031} C_VEL
LIN {X 0,Y 410.496,Z 268.394,A -85,B 0,C 180,E1 -10373.19,E2 -10373.19} C_VEL
LIN {X 0,Y 410.606,Z 265.506,A -85,B 0,C 180,E1 -10375.335,E2 -10375.335} C_VEL
LIN {X 0,Y 410.775,Z 261.268,A -85,B 0,C 180,E1 -10378.624,E2 -10378.624} C_VEL
LIN {X 0,Y 410.951,Z 256.976,A -85,B 0,C 180,E1 -10382.016,E2 -10382.016} C_VEL
LIN {X 0,Y 411.084,Z 253.488,A -85,B 0,C 180,E1 -10384.853,E2 -10384.853} C_VEL
LIN {X 0,Y 411.074,Z 252.659,A -85,B 0,C 180,E1 -10385.541,E2 -10385.541} C_VEL
LIN {X 0,Y 411.158,Z 252.273,A -85,B 0,C 180,E1 -10386.746,E2 -10386.746} C_VEL
LIN {X 0,Y 411.171,Z 252.265,A -85,B 0,C 180,E1 -10389.72,E2 -10389.72} C_VEL
LIN {X 0,Y 411.164,Z 252.267,A -85,B 0,C 180,E1 -10393.135,E2 -10393.135} C_VEL
LIN {X 0,Y 411.169,Z 252.268,A -85,B 0,C 180,E1 -10395.881,E2 -10395.881} C_VEL
LIN {X 0,Y 411.163,Z 252.269,A -85,B 0,C 180,E1 -10398.772,E2 -10398.772} C_VEL
LIN {X 0,Y 411.193,Z 252.267,A -85,B 0,C 180,E1 -10402.026,E2 -10402.026} C_VEL
LIN {X 0,Y 411.207,Z 252.263,A -85,B 0,C 180,E1 -10405.666,E2 -10405.666} C_VEL
LIN {X 0,Y 411.192,Z 252.264,A -85,B 0,C 180,E1 -10409.152,E2 -10409.152} C_VEL
LIN {X 0,Y 411.262,Z 252.255,A -85,B 0,C 180,E1 -10412.522,E2 -10412.522} C_VEL
LIN {X 0,Y 411.223,Z 252.264,A -85,B 0,C 180,E1 -10415.784,E2 -10415.784} C_VEL
LIN {X 0,Y 411.199,Z 252.263,A -85,B 0,C 180,E1 -10418.966,E2 -10418.966} C_VEL
LIN {X 0,Y 411.246,Z 252.257,A -85,B 0,C 180,E1 -10422.085,E2 -10422.085} C_VEL
LIN {X 0,Y 411.259,Z 252.259,A -85,B 0,C 180,E1 -10425.147,E2 -10425.147} C_VEL
LIN {X 0,Y 411.287,Z 252.252,A -85,B 0,C 180,E1 -10428.167,E2 -10428.167} C_VEL
LIN {X 0,Y 411.441,Z 252.232,A -85,B 0,C 180,E1 -10432.192,E2 -10432.192} C_VEL
LIN {X 0,Y 411.448,Z 252.23,A -85,B 0,C 180,E1 -10434.118,E2 -10434.118} C_VEL
LIN {X 0,Y 411.508,Z 252.224,A -85,B 0,C 180,E1 -10438.042,E2 -10438.042} C_VEL
LIN {X 0,Y 411.448,Z 252.235,A -85,B 0,C 180,E1 -10440.979,E2 -10440.979} C_VEL
LIN {X 0,Y 411.46,Z 252.234,A -85,B 0,C 180,E1 -10442.937,E2 -10442.937} C_VEL
LIN {X 0,Y 411.47,Z 252.229,A -85,B 0,C 180,E1 -10445.882,E2 -10445.882} C_VEL
LIN {X 0,Y 411.315,Z 252.249,A -85,B 0,C 180,E1 -10448.846,E2 -10448.846} C_VEL
LIN {X 0,Y 411.276,Z 252.254,A -85,B 0,C 180,E1 -10451.833,E2 -10451.833} C_VEL
LIN {X 0,Y 411.262,Z 252.256,A -85,B 0,C 180,E1 -10454.853,E2 -10454.853} C_VEL
LIN {X 0,Y 411.256,Z 252.259,A -85,B 0,C 180,E1 -10457.915,E2 -10457.915} C_VEL
LIN {X 0,Y 411.199,Z 252.262,A -85,B 0,C 180,E1 -10461.034,E2 -10461.034} C_VEL
LIN {X 0,Y 411.194,Z 252.265,A -85,B 0,C 180,E1 -10464.217,E2 -10464.217} C_VEL
LIN {X 0,Y 411.19,Z 252.266,A -85,B 0,C 180,E1 -10467.483,E2 -10467.483} C_VEL
LIN {X 0,Y 411.191,Z 252.264,A -85,B 0,C 180,E1 -10470.848,E2 -10470.848} C_VEL
LIN {X 0,Y 411.208,Z 252.262,A -85,B 0,C 180,E1 -10474.333,E2 -10474.333} C_VEL
